LIN {X 0,Y 234.64,Z 487.256,A -85,B 0,C 180,E1 -19654.688,E2 -19654.688} C_VEL
LIN {X 0,Y 234.89,Z 487.224,A -85,B 0,C 180,E1 -19658.928,E2 -19658.928} C_VEL
LIN {X 0,Y 234.891,Z 487.223,A -85,B 0,C 180,E1 -19663.486,E2 -19663.486} C_VEL
LIN {X 0,Y 234.891,Z 487.226,A -85,B 0,C 180,E1 -19666.514,E2 -19666.514} C_VEL
LIN {X 0,Y 234.959,Z 487.213,A -85,B 0,C 180,E1 -19671.086,E2 -19671.086} C_VEL
LIN {X 0,Y 234.964,Z 487.215,A -85,B 0,C 180,E1 -19675.367,E2 -19675.367} C_VEL
LIN {X 0,Y 234.973,Z 487.214,A -85,B 0,C 180,E1 -19680.158,E2 -19680.158} C_VEL
LIN {X 0,Y 234.998,Z 487.212,A -85,B 0,C 180,E1 -19683.794,E2 -19683.794} C_VEL
LIN {X 0,Y 235.016,Z 487.206,A -85,B 0,C 180,E1 -19688.97,E2 -19688.97} C_VEL
LIN {X 0,Y 235.101,Z 487.198,A -85,B 0,C 180,E1 -19693.059,E2 -19693.059} C_VEL
LIN {X 0,Y 235.12,Z 487.195,A -85,B 0,C 180,E1 -19697.922,E2 -19697.922} C_VEL
LIN {X 0,Y 235.336,Z 487.169,A -85,B 0,C 180,E1 -19701.412,E2 -19701.412} C_VEL
LIN {X 0,Y 235.378,Z 487.163,A -85,B 0,C 180,E1 -19703.14,E2 -19703.14} C_VEL
LIN {X 0,Y 235.6,Z 487.138,A -85,B 0,C 180,E1 -19708.29,E2 -19708.29} C_VEL
LIN {X 0,Y 235.6,Z 487.138,A -85,B 0,C 180,E1 -19711.709,E2 -19711.709} C_VEL
LIN {X 0,Y 235.364,Z 487.164,A -85,B 0,C 180,E1 -19716.859,E2 -19716.859} C_VEL
LIN {X 0,Y 235.218,Z 487.184,A -85,B 0,C 180,E1 -19720.327,E2 -19720.327} C_VEL
LIN {X 0,Y 235.118,Z 487.196,A -85,B 0,C 180,E1 -19725.606,E2 -19725.606} C_VEL
LIN {X 0,Y 235.013,Z 487.209,A -85,B 0,C 180,E1 -19729.205,E2 -19729.205} C_VEL
LIN {X 0,Y 234.965,Z 487.212,A -85,B 0,C 180,E1 -19732.882,E2 -19732.882} C_VEL
LIN {X 0,Y 234.972,Z 487.214,A -85,B 0,C 180,E1 -19736.657,E2 -19736.657} C_VEL
LIN {X 0,Y 234.934,Z 487.215,A -85,B 0,C 180,E1 -19740.567,E2 -19740.567} C_VEL
LIN {X 0,Y 234.963,Z 487.215,A -85,B 0,C 180,E1 -19744.632,E2 -19744.632} C_VEL
LIN {X 0,Y 234.944,Z 487.215,A -85,B 0,C 180,E1 -19748.944,E2 -19748.944} C_VEL
LIN {X 0,Y 234.889,Z 487.226,A -85,B 0,C 180,E1 -19753.485,E2 -19753.485} C_VEL
LIN {X 0,Y 234.889,Z 487.223,A -85,B 0,C 180,E1 -19756.513,E2 -19756.513} C_VEL
LIN {X 0,Y 234.92,Z 487.22,A -85,B 0,C 180,E1 -19761.078,E2 -19761.078} C_VEL
LIN {X 0,Y 234.943,Z 487.219,A -85,B 0,C 180,E1 -19765.363,E2 -19765.363} C_VEL
LIN {X 0,Y 234.933,Z 487.22,A -85,B 0,C 180,E1 -19769.432,E2 -19769.432} C_VEL
LIN {X 0,Y 234.995,Z 487.212,A -85,B 0,C 180,E1 -19773.793,E2 -19773.793} C_VEL
LIN {X 0,Y 235.013,Z 487.209,A -85,B 0,C 180,E1 -19778.969,E2 -19778.969} C_VEL
LIN {X 0,Y 235.097,Z 487.198,A -85,B 0,C 180,E1 -19783.059,E2 -19783.059} C_VEL
LIN {X 0,Y 235.148,Z 487.194,A -85,B 0,C 180,E1 -19787.923,E2 -19787.923} C_VEL
LIN {X 0,Y 235.391,Z 487.164,A -85,B 0,C 180,E1 -19791.414,E2 -19791.414} C_VEL
LIN {X 0,Y 235.407,Z 487.159,A -85,B 0,C 180,E1 -19793.141,E2 -19793.141} C_VEL
LIN {X 0,Y 235.597,Z 487.136,A -85,B 0,C 180,E1 -19798.29,E2 -19798.29} C_VEL
LIN {X 0,Y 235.597,Z 487.136,A -85,B 0,C 180,E1 -19801.709,E2 -19801.709} C_VEL
LIN {X 0,Y 235.406,Z 487.16,A -85,B 0,C 180,E1 -19806.858,E2 -19806.858} C_VEL
LIN {X 0,Y 235.253,Z 487.176,A -85,B 0,C 180,E1 -19810.325,E2 -19810.325} C_VEL
LIN {X 0,Y 235.114,Z 487.199,A -85,B 0,C 180,E1 -19815.606,E2 -19815.606} C_VEL
LIN {X 0,Y 235.009,Z 487.21,A -85,B 0,C 180,E1 -19819.205,E2 -19819.205} C_VEL
LIN {X 0,Y 234.961,Z 487.216,A -85,B 0,C 180,E1 -19822.883,E2 -19822.883} C_VEL
LIN {X 0,Y 234.967,Z 487.214,A -85,B 0,C 180,E1 -19826.657,E2 -19826.657} C_VEL
LIN {X 0,Y 234.922,Z 487.219,A -85,B 0,C 180,E1 -19830.569,E2 -19830.569} C_VEL
LIN {X 0,Y 234.96,Z 487.215,A -85,B 0,C 180,E1 -19834.633,E2 -19834.633} C_VEL
LIN {X 0,Y 234.966,Z 487.214,A -85,B 0,C 180,E1 -19838.952,E2 -19838.952} C_VEL
LIN {X 0,Y 235.159,Z 487.364,A -85,B 0,C 180,E1 -19843.423,E2 -19843.423} C_VEL
LIN {X 0,Y 236.059,Z 492.395,A -85,B 0,C 180,E1 -19848.099,E2 -19848.099} C_VEL
LIN {X 0,Y 236.71,Z 496.121,A -85,B 0,C 180,E1 -19851.428,E2 -19851.428} C_VEL
LIN {X 0,Y 236.891,Z 498.627,A -85,B 0,C 180,E1 -19853.605,E2 -19853.605} C_VEL
LIN {X 0,Y 236.198,Z 501.988,A -85,B 0,C 180,E1 -19856.422,E2 -19856.422} C_VEL
LIN {X 0,Y 234.967,Z 507.976,A -85,B 0,C 180,E1 -19861.408,E2 -19861.408} C_VEL
LIN {X 0,Y 234.627,Z 509.787,A -85,B 0,C 180,E1 -19862.901,E2 -19862.901} C_VEL
LIN {X 0,Y 234.164,Z 511.237,A -85,B 0,C 180,E1 -19863.76,E2 -19863.76} C_VEL
LIN {X 0,Y 232.71,Z 514.431,A -85,B 0,C 180,E1 -19864.89,E2 -19864.89} C_VEL
LIN {X 0,Y 230.881,Z 518.451,A -85,B 0,C 180,E1 -19865.841,E2 -19865.841} C_VEL
LIN {X 0,Y 228.657,Z 524.846,A -85,B 0,C 180,E1 -19866.905,E2 -19866.905} C_VEL
LIN {X 0,Y 227.893,Z 530.135,A -85,B 0,C 180,E1 -19867.569,E2 -19867.569} C_VEL
LIN {X 0,Y 227.932,Z 531.961,A -85,B 0,C 180,E1 -19867.766,E2 -19867.766} C_VEL
LIN {X 0,Y 228.995,Z 545.084,A -85,B 0,C 180,E1 -19869.333,E2 -19869.333} C_VEL
LIN {X 0,Y 230.354,Z 558.222,A -85,B 0,C 180,E1 -19871.293,E2 -19871.293} C_VEL
LIN {X 0,Y 229.91,Z 564.614,A -85,B 0,C 180,E1 -19872.431,E2 -19872.431} C_VEL
LIN {X 0,Y 228.743,Z 574.152,A -85,B 0,C 180,E1 -19874.405,E2 -19874.405} C_VEL
LIN {X 0,Y 227.85,Z 583.066,A -85,B 0,C 180,E1 -19876.625,E2 -19876.625} C_VEL
LIN {X 0,Y 227.058,Z 591.816,A -85,B 0,C 180,E1 -19879.298,E2 -19879.298} C_VEL
LIN {X 0,Y 226.683,Z 598.895,A -85,B 0,C 180,E1 -19881.981,E2 -19881.981} C_VEL
LIN {X 0,Y 226.508,Z 604.521,A -85,B 0,C 180,E1 -19884.659,E2 -19884.659} C_VEL
LIN {X 0,Y 226.501,Z 608.915,A -85,B 0,C 180,E1 -19887.333,E2 -19887.333} C_VEL
LIN {X 0,Y 226.588,Z 612.194,A -85,B 0,C 180,E1 -19890,E2 -19890} C_VEL
LIN {X 0,Y 226.285,Z 613.769,A -85,B 0,C 180,E1 -19891.78,E2 -19891.78} C_VEL
LIN {X 0,Y 225.922,Z 615.651,A -85,B 0,C 180,E1 -19895.355,E2 -19895.355} C_VEL
LIN {X 0,Y 226.153,Z 616.056,A -85,B 0,C 180,E1 -19898.939,E2 -19898.939} C_VEL
LIN {X 0,Y 227.195,Z 615.063,A -85,B 0,C 180,E1 -19902.506,E2 -19902.506} C_VEL
LIN {X 0,Y 229.251,Z 612.694,A -85,B 0,C 180,E1 -19906.017,E2 -19906.017} C_VEL
LIN {X 0,Y 232.384,Z 608.934,A -85,B 0,C 180,E1 -19909.432,E2 -19909.432} C_VEL
LIN {X 0,Y 236.369,Z 603.761,A -85,B 0,C 180,E1 -19912.739,E2 -19912.739} C_VEL
LIN {X 0,Y 240.175,Z 598.876,A -85,B 0,C 180,E1 -19915.107,E2 -19915.107} C_VEL
LIN {X 0,Y 246.115,Z 590.937,A -85,B 0,C 180,E1 -19918.111,E2 -19918.111} C_VEL
LIN {X 0,Y 251.032,Z 583.774,A -85,B 0,C 180,E1 -19920.261,E2 -19920.261} C_VEL
LIN {X 0,Y 253.685,Z 578.77,A -85,B 0,C 180,E1 -19921.761,E2 -19921.761} C_VEL
LIN {X 0,Y 256.161,Z 572.028,A -85,B 0,C 180,E1 -19923.971,E2 -19923.971} C_VEL
LIN {X 0,Y 258.198,Z 564.336,A -85,B 0,C 180,E1 -19926.786,E2 -19926.786} C_VEL
LIN {X 0,Y 259.165,Z 560.003,A -85,B 0,C 180,E1 -19928.588,E2 -19928.588} C_VEL
LIN {X 0,Y 259.899,Z 556.273,A -85,B 0,C 180,E1 -19930.466,E2 -19930.466} C_VEL
LIN {X 0,Y 260.12,Z 553.505,A -85,B 0,C 180,E1 -19932.49,E2 -19932.49} C_VEL
LIN {X 0,Y 260.395,Z 551.497,A -85,B 0,C 180,E1 -19934.567,E2 -19934.567} C_VEL
LIN {X 0,Y 260.509,Z 550.609,A -85,B 0,C 180,E1 -19936.754,E2 -19936.754} C_VEL
LIN {X 0,Y 260.631,Z 551.068,A -85,B 0,C 180,E1 -19939.672,E2 -19939.672} C_VEL
LIN {X 0,Y 260.998,Z 552.105,A -85,B 0,C 180,E1 -19941.733,E2 -19941.733} C_VEL
LIN {X 0,Y 261.38,Z 553.873,A -85,B 0,C 180,E1 -19943.77,E2 -19943.77} C_VEL
LIN {X 0,Y 261.44,Z 557.559,A -85,B 0,C 180,E1 -19946.444,E2 -19946.444} C_VEL
LIN {X 0,Y 260.967,Z 561.356,A -85,B 0,C 180,E1 -19948.526,E2 -19948.526} C_VEL
LIN {X 0,Y 260.113,Z 563.075,A -85,B 0,C 180,E1 -19949.112,E2 -19949.112} C_VEL
LIN {X 0,Y 253.924,Z 571.515,A -85,B 0,C 180,E1 -19951.482,E2 -19951.482} C_VEL
LIN {X 0,Y 248.247,Z 578.439,A -85,B 0,C 180,E1 -19953.972,E2 -19953.972} C_VEL
LIN {X 0,Y 243.868,Z 583.268,A -85,B 0,C 180,E1 -19956.205,E2 -19956.205} C_VEL
LIN {X 0,Y 238.859,Z 588.281,A -85,B 0,C 180,E1 -19959.325,E2 -19959.325} C_VEL
LIN {X 0,Y 234.733,Z 591.746,A -85,B 0,C 180,E1 -19962.579,E2 -19962.579} C_VEL
LIN {X 0,Y 232.898,Z 592.963,A -85,B 0,C 180,E1 -19964.242,E2 -19964.242} C_VEL
LIN {X 0,Y 230.124,Z 594.323,A -85,B 0,C 180,E1 -19967.656,E2 -19967.656} C_VEL
LIN {X 0,Y 227.906,Z 594.264,A -85,B 0,C 180,E1 -19971.131,E2 -19971.131} C_VEL
LIN {X 0,Y 226.816,Z 592.766,A -85,B 0,C 180,E1 -19974.667,E2 -19974.667} C_VEL
LIN {X 0,Y 226.416,Z 591.482,A -85,B 0,C 180,E1 -19976.441,E2 -19976.441} C_VEL
LIN {X 0,Y 225.976,Z 587.71,A -85,B 0,C 180,E1 -19980,E2 -19980} C_VEL
LIN {X 0,Y 225.999,Z 583.818,A -85,B 0,C 180,E1 -19982.674,E2 -19982.674} C_VEL
LIN {X 0,Y 226.077,Z 578.823,A -85,B 0,C 180,E1 -19985.352,E2 -19985.352} C_VEL
LIN {X 0,Y 226.624,Z 571.523,A -85,B 0,C 180,E1 -19988.471,E2 -19988.471} C_VEL
LIN {X 0,Y 227.301,Z 563.747,A -85,B 0,C 180,E1 -19991.143,E2 -19991.143} C_VEL
LIN {X 0,Y 228.272,Z 554.253,A -85,B 0,C 180,E1 -19993.805,E2 -19993.805} C_VEL
LIN {X 0,Y 229.552,Z 543.626,A -85,B 0,C 180,E1 -19996.223,E2 -19996.223} C_VEL
LIN {X 0,Y 230.933,Z 531.732,A -85,B 0,C 180,E1 -19998.406,E2 -19998.406} C_VEL
LIN {X 0,Y 232.048,Z 520.174,A -85,B 0,C 180,E1 -20000.133,E2 -20000.133} C_VEL
LIN {X 0,Y 229.504,Z 506.121,A -85,B 0,C 180,E1 -20001.896,E2 -20001.896} C_VEL
LIN {X 0,Y 227.192,Z 492.743,A -85,B 0,C 180,E1 -20003.213,E2 -20003.213} C_VEL
LIN {X 0,Y 226.512,Z 488.273,A -85,B 0,C 180,E1 -20003.585,E2 -20003.585} C_VEL
LIN {X 0,Y 226.902,Z 488.224,A -85,B 0,C 180,E1 -20007.685,E2 -20007.685} C_VEL
LIN {X 0,Y 227.31,Z 488.167,A -85,B 0,C 180,E1 -20011.71,E2 -20011.71} C_VEL
LIN {X 0,Y 227.698,Z 488.121,A -85,B 0,C 180,E1 -20015.906,E2 -20015.906} C_VEL
LIN {X 0,Y 227.817,Z 488.105,A -85,B 0,C 180,E1 -20019.535,E2 -20019.535} C_VEL
LIN {X 0,Y 227.812,Z 488.105,A -85,B 0,C 180,E1 -20022.743,E2 -20022.743} C_VEL
LIN {X 0,Y 227.818,Z 488.105,A -85,B 0,C 180,E1 -20027.259,E2 -20027.259} C_VEL
LIN {X 0,Y 227.873,Z 488.098,A -85,B 0,C 180,E1 -20031.914,E2 -20031.914} C_VEL
LIN {X 0,Y 227.893,Z 488.097,A -85,B 0,C 180,E1 -20036.373,E2 -20036.373} C_VEL
LIN {X 0,Y 227.923,Z 488.093,A -85,B 0,C 180,E1 -20040.438,E2 -20040.438} C_VEL
LIN {X 0,Y 227.933,Z 488.092,A -85,B 0,C 180,E1 -20044.426,E2 -20044.426} C_VEL
LIN {X 0,Y 227.967,Z 488.087,A -85,B 0,C 180,E1 -20048.287,E2 -20048.287} C_VEL
LIN {X 0,Y 228.04,Z 488.078,A -85,B 0,C 180,E1 -20052.825,E2 -20052.825} C_VEL
LIN {X 0,Y 228.078,Z 488.07,A -85,B 0,C 180,E1 -20057.543,E2 -20057.543} C_VEL
LIN {X 0,Y 228.272,Z 488.048,A -85,B 0,C 180,E1 -20061.144,E2 -20061.144} C_VEL
LIN {X 0,Y 228.329,Z 488.041,A -85,B 0,C 180,E1 -20062.927,E2 -20062.927} C_VEL
LIN {X 0,Y 228.559,Z 488.015,A -85,B 0,C 180,E1 -20068.238,E2 -20068.238} C_VEL
LIN {X 0,Y 228.558,Z 488.015,A -85,B 0,C 180,E1 -20071.762,E2 -20071.762} C_VEL
LIN {X 0,Y 228.316,Z 488.042,A -85,B 0,C 180,E1 -20077.072,E2 -20077.072} C_VEL
LIN {X 0,Y 228.15,Z 488.063,A -85,B 0,C 180,E1 -20080.651,E2 -20080.651} C_VEL
LIN {X 0,Y 228.069,Z 488.074,A -85,B 0,C 180,E1 -20084.271,E2 -20084.271} C_VEL
LIN {X 0,Y 228.007,Z 488.085,A -85,B 0,C 180,E1 -20087.953,E2 -20087.953} C_VEL
LIN {X 0,Y 227.934,Z 488.089,A -85,B 0,C 180,E1 -20092.329,E2 -20092.329} C_VEL
LIN {X 0,Y 227.946,Z 488.089,A -85,B 0,C 180,E1 -20096.602,E2 -20096.602} C_VEL
LIN {X 0,Y 227.911,Z 488.091,A -85,B 0,C 180,E1 -20100.295,E2 -20100.295} C_VEL
LIN {X 0,Y 227.893,Z 488.098,A -85,B 0,C 180,E1 -20103.717,E2 -20103.717} C_VEL
LIN {X 0,Y 227.872,Z 488.098,A -85,B 0,C 180,E1 -20108.085,E2 -20108.085} C_VEL
LIN {X 0,Y 227.816,Z 488.105,A -85,B 0,C 180,E1 -20112.741,E2 -20112.741} C_VEL
LIN {X 0,Y 227.812,Z 488.105,A -85,B 0,C 180,E1 -20117.257,E2 -20117.257} C_VEL
LIN {X 0,Y 227.846,Z 488.104,A -85,B 0,C 180,E1 -20121.908,E2 -20121.908} C_VEL
LIN {X 0,Y 227.884,Z 488.094,A -85,B 0,C 180,E1 -20126.375,E2 -20126.375} C_VEL
LIN {X 0,Y 227.921,Z 488.092,A -85,B 0,C 180,E1 -20130.437,E2 -20130.437} C_VEL
LIN {X 0,Y 227.93,Z 488.089,A -85,B 0,C 180,E1 -20134.425,E2 -20134.425} C_VEL
LIN {X 0,Y 227.963,Z 488.087,A -85,B 0,C 180,E1 -20138.287,E2 -20138.287} C_VEL
LIN {X 0,Y 228.036,Z 488.077,A -85,B 0,C 180,E1 -20142.825,E2 -20142.825} C_VEL
LIN {X 0,Y 228.095,Z 488.073,A -85,B 0,C 180,E1 -20147.544,E2 -20147.544} C_VEL
LIN {X 0,Y 228.326,Z 488.043,A -85,B 0,C 180,E1 -20151.146,E2 -20151.146} C_VEL
LIN {X 0,Y 228.359,Z 488.036,A -85,B 0,C 180,E1 -20152.928,E2 -20152.928} C_VEL
LIN {X 0,Y 228.556,Z 488.013,A -85,B 0,C 180,E1 -20158.237,E2 -20158.237} C_VEL
LIN {X 0,Y 228.555,Z 488.012,A -85,B 0,C 180,E1 -20161.762,E2 -20161.762} C_VEL
LIN {X 0,Y 228.359,Z 488.039,A -85,B 0,C 180,E1 -20167.071,E2 -20167.071} C_VEL
LIN {X 0,Y 228.172,Z 488.058,A -85,B 0,C 180,E1 -20170.65,E2 -20170.65} C_VEL
LIN {X 0,Y 228.058,Z 488.075,A -85,B 0,C 180,E1 -20176.102,E2 -20176.102} C_VEL
LIN {X 0,Y 227.943,Z 488.088,A -85,B 0,C 180,E1 -20179.825,E2 -20179.825} C_VEL
LIN {X 0,Y 227.914,Z 488.095,A -85,B 0,C 180,E1 -20183.632,E2 -20183.632} C_VEL
LIN {X 0,Y 227.879,Z 488.097,A -85,B 0,C 180,E1 -20187.556,E2 -20187.556} C_VEL
LIN {X 0,Y 227.869,Z 488.101,A -85,B 0,C 180,E1 -20191.622,E2 -20191.622} C_VEL
LIN {X 0,Y 227.901,Z 488.093,A -85,B 0,C 180,E1 -20195.868,E2 -20195.868} C_VEL
LIN {X 0,Y 227.916,Z 488.092,A -85,B 0,C 180,E1 -20200.357,E2 -20200.357} C_VEL
LIN {X 0,Y 228.11,Z 488.177,A -85,B 0,C 180,E1 -20203.428,E2 -20203.428} C_VEL
LIN {X 0,Y 229.108,Z 493.726,A -85,B 0,C 180,E1 -20208.737,E2 -20208.737} C_VEL
LIN {X 0,Y 229.739,Z 497.598,A -85,B 0,C 180,E1 -20212.279,E2 -20212.279} C_VEL
LIN {X 0,Y 229.664,Z 500.056,A -85,B 0,C 180,E1 -20214.45,E2 -20214.45} C_VEL
LIN {X 0,Y 228.276,Z 505.955,A -85,B 0,C 180,E1 -20219.546,E2 -20219.546} C_VEL
LIN {X 0,Y 227.217,Z 511.521,A -85,B 0,C 180,E1 -20224.34,E2 -20224.34} C_VEL
LIN {X 0,Y 226.937,Z 513.601,A -85,B 0,C 180,E1 -20226.139,E2 -20226.139} C_VEL
LIN {X 0,Y 227.507,Z 526.824,A -85,B 0,C 180,E1 -20227.248,E2 -20227.248} C_VEL
LIN {X 0,Y 227.932,Z 531.961,A -85,B 0,C 180,E1 -20227.766,E2 -20227.766} C_VEL
LIN {X 0,Y 227.751,Z 537.377,A -85,B 0,C 180,E1 -20228.353,E2 -20228.353} C_VEL
LIN {X 0,Y 225.867,Z 546.084,A -85,B 0,C 180,E1 -20229.434,E2 -20229.434} C_VEL
LIN {X 0,Y 224.113,Z 552.813,A -85,B 0,C 180,E1 -20230.42,E2 -20230.42} C_VEL
LIN {X 0,Y 223.29,Z 559.395,A -85,B 0,C 180,E1 -20231.529,E2 -20231.529} C_VEL
LIN {X 0,Y 222.075,Z 570.338,A -85,B 0,C 180,E1 -20233.688,E2 -20233.688} C_VEL
LIN {X 0,Y 221.162,Z 578.904,A -85,B 0,C 180,E1 -20235.743,E2 -20235.743} C_VEL
LIN {X 0,Y 220.241,Z 588.254,A -85,B 0,C 180,E1 -20238.496,E2 -20238.496} C_VEL
LIN {X 0,Y 219.779,Z 595.885,A -85,B 0,C 180,E1 -20241.264,E2 -20241.264} C_VEL
LIN {X 0,Y 219.564,Z 601.199,A -85,B 0,C 180,E1 -20243.626,E2 -20243.626} C_VEL
LIN {X 0,Y 219.505,Z 606.125,A -85,B 0,C 180,E1 -20246.329,E2 -20246.329} C_VEL
LIN {X 0,Y 219.528,Z 609.978,A -85,B 0,C 180,E1 -20249.083,E2 -20249.083} C_VEL
LIN {X 0,Y 219.571,Z 611.024,A -85,B 0,C 180,E1 -20250,E2 -20250} C_VEL
LIN {X 0,Y 219.273,Z 612.679,A -85,B 0,C 180,E1 -20251.837,E2 -20251.837} C_VEL
LIN {X 0,Y 218.886,Z 614.828,A -85,B 0,C 180,E1 -20255.528,E2 -20255.528} C_VEL
LIN {X 0,Y 219.122,Z 615.516,A -85,B 0,C 180,E1 -20259.229,E2 -20259.229} C_VEL
LIN {X 0,Y 220.227,Z 614.78,A -85,B 0,C 180,E1 -20262.909,E2 -20262.909} C_VEL
LIN {X 0,Y 222.43,Z 612.714,A -85,B 0,C 180,E1 -20266.522,E2 -20266.522} C_VEL
LIN {X 0,Y 225.697,Z 609.304,A -85,B 0,C 180,E1 -20270.032,E2 -20270.032} C_VEL
LIN {X 0,Y 228.769,Z 605.774,A -85,B 0,C 180,E1 -20272.65,E2 -20272.65} C_VEL
LIN {X 0,Y 233.847,Z 599.995,A -85,B 0,C 180,E1 -20275.835,E2 -20275.835} C_VEL
LIN {X 0,Y 240.003,Z 592.536,A -85,B 0,C 180,E1 -20278.893,E2 -20278.893} C_VEL
LIN {X 0,Y 245.955,Z 584.69,A -85,B 0,C 180,E1 -20281.432,E2 -20281.432} C_VEL
LIN {X 0,Y 248.034,Z 581.14,A -85,B 0,C 180,E1 -20282.573,E2 -20282.573} C_VEL
LIN {X 0,Y 251.092,Z 574.057,A -85,B 0,C 180,E1 -20285.116,E2 -20285.116} C_VEL
LIN {X 0,Y 253.186,Z 567.758,A -85,B 0,C 180,E1 -20287.639,E2 -20287.639} C_VEL
LIN {X 0,Y 254.692,Z 562.719,A -85,B 0,C 180,E1 -20289.973,E2 -20289.973} C_VEL
LIN {X 0,Y 255.329,Z 559.621,A -85,B 0,C 180,E1 -20291.997,E2 -20291.997} C_VEL
LIN {X 0,Y 255.734,Z 557.187,A -85,B 0,C 180,E1 -20294.396,E2 -20294.396} C_VEL
LIN {X 0,Y 255.891,Z 556.401,A -85,B 0,C 180,E1 -20295.569,E2 -20295.569} C_VEL
LIN {X 0,Y 255.916,Z 556.066,A -85,B 0,C 180,E1 -20297.858,E2 -20297.858} C_VEL
LIN {X 0,Y 256.097,Z 556.948,A -85,B 0,C 180,E1 -20300.863,E2 -20300.863} C_VEL
LIN {X 0,Y 256.424,Z 559.105,A -85,B 0,C 180,E1 -20303.786,E2 -20303.786} C_VEL
LIN {X 0,Y 256.22,Z 561.053,A -85,B 0,C 180,E1 -20305.376,E2 -20305.376} C_VEL
LIN {X 0,Y 255.688,Z 564.505,A -85,B 0,C 180,E1 -20307.604,E2 -20307.604} C_VEL
LIN {X 0,Y 254.553,Z 566.48,A -85,B 0,C 180,E1 -20308.361,E2 -20308.361} C_VEL
LIN {X 0,Y 248.104,Z 574.414,A -85,B 0,C 180,E1 -20310.749,E2 -20310.749} C_VEL
LIN {X 0,Y 242.187,Z 580.835,A -85,B 0,C 180,E1 -20313.27,E2 -20313.27} C_VEL
LIN {X 0,Y 237.65,Z 585.299,A -85,B 0,C 180,E1 -20315.543,E2 -20315.543} C_VEL
LIN {X 0,Y 232.418,Z 589.853,A -85,B 0,C 180,E1 -20318.724,E2 -20318.724} C_VEL
LIN {X 0,Y 228.076,Z 592.969,A -85,B 0,C 180,E1 -20322.053,E2 -20322.053} C_VEL
LIN {X 0,Y 226.164,Z 594.008,A -85,B 0,C 180,E1 -20323.76,E2 -20323.76} C_VEL
LIN {X 0,Y 223.231,Z 595.007,A -85,B 0,C 180,E1 -20327.269,E2 -20327.269} C_VEL
LIN {X 0,Y 220.919,Z 594.665,A -85,B 0,C 180,E1 -20330.848,E2 -20330.848} C_VEL
LIN {X 0,Y 219.754,Z 592.868,A -85,B 0,C 180,E1 -20334.495,E2 -20334.495} C_VEL
LIN {X 0,Y 219.052,Z 589.599,A -85,B 0,C 180,E1 -20338.162,E2 -20338.162} C_VEL
LIN {X 0,Y 218.882,Z 586.103,A -85,B 0,C 180,E1 -20340.92,E2 -20340.92} C_VEL
LIN {X 0,Y 218.927,Z 581.625,A -85,B 0,C 180,E1 -20343.682,E2 -20343.682} C_VEL
LIN {X 0,Y 219.256,Z 575.022,A -85,B 0,C 180,E1 -20346.904,E2 -20346.904} C_VEL
LIN {X 0,Y 219.771,Z 567.895,A -85,B 0,C 180,E1 -20349.666,E2 -20349.666} C_VEL
LIN {X 0,Y 220.639,Z 559.205,A -85,B 0,C 180,E1 -20352.416,E2 -20352.416} C_VEL
LIN {X 0,Y 221.802,Z 548.64,A -85,B 0,C 180,E1 -20355.154,E2 -20355.154} C_VEL
LIN {X 0,Y 223.056,Z 537.863,A -85,B 0,C 180,E1 -20357.418,E2 -20357.418} C_VEL
LIN {X 0,Y 224.215,Z 527.534,A -85,B 0,C 180,E1 -20359.216,E2 -20359.216} C_VEL
LIN {X 0,Y 224.842,Z 520.022,A -85,B 0,C 180,E1 -20360.325,E2 -20360.325} C_VEL
LIN {X 0,Y 222.45,Z 506.821,A -85,B 0,C 180,E1 -20362.035,E2 -20362.035} C_VEL
LIN {X 0,Y 220.202,Z 493.731,A -85,B 0,C 180,E1 -20363.374,E2 -20363.374} C_VEL
LIN {X 0,Y 219.505,Z 489.147,A -85,B 0,C 180,E1 -20363.777,E2 -20363.777} C_VEL
LIN {X 0,Y 219.951,Z 489.087,A -85,B 0,C 180,E1 -20368.64,E2 -20368.64} C_VEL
LIN {X 0,Y 220.361,Z 489.031,A -85,B 0,C 180,E1 -20372.833,E2 -20372.833} C_VEL
LIN {X 0,Y 220.711,Z 488.99,A -85,B 0,C 180,E1 -20377.243,E2 -20377.243} C_VEL
LIN {X 0,Y 220.776,Z 488.984,A -85,B 0,C 180,E1 -20380.182,E2 -20380.182} C_VEL
LIN {X 0,Y 220.777,Z 488.985,A -85,B 0,C 180,E1 -20384.454,E2 -20384.454} C_VEL
LIN {X 0,Y 220.779,Z 488.984,A -85,B 0,C 180,E1 -20388.049,E2 -20388.049} C_VEL
LIN {X 0,Y 220.835,Z 488.975,A -85,B 0,C 180,E1 -20392.794,E2 -20392.794} C_VEL
LIN {X 0,Y 220.828,Z 488.975,A -85,B 0,C 180,E1 -20397.245,E2 -20397.245} C_VEL
LIN {X 0,Y 220.84,Z 488.973,A -85,B 0,C 180,E1 -20401.486,E2 -20401.486} C_VEL
LIN {X 0,Y 220.872,Z 488.971,A -85,B 0,C 180,E1 -20405.565,E2 -20405.565} C_VEL
LIN {X 0,Y 220.898,Z 488.965,A -85,B 0,C 180,E1 -20409.514,E2 -20409.514} C_VEL
LIN {X 0,Y 221.021,Z 488.952,A -85,B 0,C 180,E1 -20413.37,E2 -20413.37} C_VEL
LIN {X 0,Y 221.086,Z 488.943,A -85,B 0,C 180,E1 -20419.004,E2 -20419.004} C_VEL
LIN {X 0,Y 221.264,Z 488.921,A -85,B 0,C 180,E1 -20422.7,E2 -20422.7} C_VEL
LIN {X 0,Y 221.517,Z 488.893,A -85,B 0,C 180,E1 -20428.181,E2 -20428.181} C_VEL
LIN {X 0,Y 221.516,Z 488.893,A -85,B 0,C 180,E1 -20431.818,E2 -20431.818} C_VEL
LIN {X 0,Y 221.253,Z 488.923,A -85,B 0,C 180,E1 -20437.299,E2 -20437.299} C_VEL
LIN {X 0,Y 221.086,Z 488.943,A -85,B 0,C 180,E1 -20440.995,E2 -20440.995} C_VEL
LIN {X 0,Y 221.021,Z 488.952,A -85,B 0,C 180,E1 -20446.629,E2 -20446.629} C_VEL
LIN {X 0,Y 220.897,Z 488.966,A -85,B 0,C 180,E1 -20450.485,E2 -20450.485} C_VEL
LIN {X 0,Y 220.871,Z 488.971,A -85,B 0,C 180,E1 -20454.434,E2 -20454.434} C_VEL
LIN {X 0,Y 220.839,Z 488.974,A -85,B 0,C 180,E1 -20458.513,E2 -20458.513} C_VEL
LIN {X 0,Y 220.827,Z 488.975,A -85,B 0,C 180,E1 -20462.754,E2 -20462.754} C_VEL
LIN {X 0,Y 220.84,Z 488.975,A -85,B 0,C 180,E1 -20467.287,E2 -20467.287} C_VEL
LIN {X 0,Y 220.777,Z 488.985,A -85,B 0,C 180,E1 -20471.951,E2 -20471.951} C_VEL
LIN {X 0,Y 220.775,Z 488.985,A -85,B 0,C 180,E1 -20475.545,E2 -20475.545} C_VEL
LIN {X 0,Y 220.808,Z 488.978,A -85,B 0,C 180,E1 -20480.462,E2 -20480.462} C_VEL
LIN {X 0,Y 220.805,Z 488.978,A -85,B 0,C 180,E1 -20485.045,E2 -20485.045} C_VEL
LIN {X 0,Y 220.869,Z 488.971,A -85,B 0,C 180,E1 -20489.394,E2 -20489.394} C_VEL
LIN {X 0,Y 220.897,Z 488.97,A -85,B 0,C 180,E1 -20493.549,E2 -20493.549} C_VEL
LIN {X 0,Y 220.879,Z 488.97,A -85,B 0,C 180,E1 -20497.553,E2 -20497.553} C_VEL
LIN {X 0,Y 220.985,Z 488.955,A -85,B 0,C 180,E1 -20502.57,E2 -20502.57} C_VEL
LIN {X 0,Y 221.027,Z 488.951,A -85,B 0,C 180,E1 -20507.139,E2 -20507.139} C_VEL
LIN {X 0,Y 221.259,Z 488.922,A -85,B 0,C 180,E1 -20510.861,E2 -20510.861} C_VEL
LIN {X 0,Y 221.312,Z 488.913,A -85,B 0,C 180,E1 -20512.702,E2 -20512.702} C_VEL
LIN {X 0,Y 221.514,Z 488.891,A -85,B 0,C 180,E1 -20518.181,E2 -20518.181} C_VEL
LIN {X 0,Y 221.513,Z 488.889,A -85,B 0,C 180,E1 -20521.818,E2 -20521.818} C_VEL
LIN {X 0,Y 221.312,Z 488.918,A -85,B 0,C 180,E1 -20527.297,E2 -20527.297} C_VEL
LIN {X 0,Y 221.117,Z 488.938,A -85,B 0,C 180,E1 -20530.994,E2 -20530.994} C_VEL
LIN {X 0,Y 221.016,Z 488.952,A -85,B 0,C 180,E1 -20536.629,E2 -20536.629} C_VEL
LIN {X 0,Y 220.893,Z 488.965,A -85,B 0,C 180,E1 -20540.486,E2 -20540.486} C_VEL
LIN {X 0,Y 220.867,Z 488.971,A -85,B 0,C 180,E1 -20544.435,E2 -20544.435} C_VEL
LIN {X 0,Y 220.826,Z 488.972,A -85,B 0,C 180,E1 -20548.515,E2 -20548.515} C_VEL
LIN {X 0,Y 220.823,Z 488.977,A -85,B 0,C 180,E1 -20552.755,E2 -20552.755} C_VEL
LIN {X 0,Y 220.838,Z 488.974,A -85,B 0,C 180,E1 -20557.288,E2 -20557.288} C_VEL
LIN {X 0,Y 220.947,Z 488.961,A -85,B 0,C 180,E1 -20561.911,E2 -20561.911} C_VEL
LIN {X 0,Y 221.085,Z 489.124,A -85,B 0,C 180,E1 -20563.599,E2 -20563.599} C_VEL
LIN {X 0,Y 221.932,Z 493.899,A -85,B 0,C 180,E1 -20568.317,E2 -20568.317} C_VEL
LIN {X 0,Y 222.644,Z 497.881,A -85,B 0,C 180,E1 -20572.106,E2 -20572.106} C_VEL
LIN {X 0,Y 222.604,Z 500.243,A -85,B 0,C 180,E1 -20574.264,E2 -20574.264} C_VEL
LIN {X 0,Y 221.199,Z 506.017,A -85,B 0,C 180,E1 -20579.446,E2 -20579.446} C_VEL
LIN {X 0,Y 220.099,Z 511.617,A -85,B 0,C 180,E1 -20584.465,E2 -20584.465} C_VEL
LIN {X 0,Y 219.849,Z 513.48,A -85,B 0,C 180,E1 -20585.948,E2 -20585.948} C_VEL
LIN {X 0,Y 220.442,Z 527.242,A -85,B 0,C 180,E1 -20587.137,E2 -20587.137} C_VEL
LIN {X 0,Y 221.545,Z 541.001,A -85,B 0,C 180,E1 -20588.726,E2 -20588.726} C_VEL
LIN {X 0,Y 222.691,Z 553.141,A -85,B 0,C 180,E1 -20590.473,E2 -20590.473} C_VEL
LIN {X 0,Y 223.29,Z 559.395,A -85,B 0,C 180,E1 -20591.529,E2 -20591.529} C_VEL
LIN {X 0,Y 222.89,Z 562.631,A -85,B 0,C 180,E1 -20592.117,E2 -20592.117} C_VEL
LIN {X 0,Y 221.851,Z 565.638,A -85,B 0,C 180,E1 -20592.714,E2 -20592.714} C_VEL
LIN {X 0,Y 218.723,Z 571.21,A -85,B 0,C 180,E1 -20593.956,E2 -20593.956} C_VEL
LIN {X 0,Y 214.845,Z 577.728,A -85,B 0,C 180,E1 -20595.68,E2 -20595.68} C_VEL
LIN {X 0,Y 213.753,Z 581.686,A -85,B 0,C 180,E1 -20596.824,E2 -20596.824} C_VEL
LIN {X 0,Y 213.012,Z 590.102,A -85,B 0,C 180,E1 -20599.545,E2 -20599.545} C_VEL
LIN {X 0,Y 212.645,Z 597.527,A -85,B 0,C 180,E1 -20602.528,E2 -20602.528} C_VEL
LIN {X 0,Y 212.526,Z 602.962,A -85,B 0,C 180,E1 -20605.258,E2 -20605.258} C_VEL
LIN {X 0,Y 212.537,Z 607.396,A -85,B 0,C 180,E1 -20608.105,E2 -20608.105} C_VEL
LIN {X 0,Y 212.572,Z 609.731,A -85,B 0,C 180,E1 -20610,E2 -20610} C_VEL
LIN {X 0,Y 212.258,Z 611.558,A -85,B 0,C 180,E1 -20611.898,E2 -20611.898} C_VEL
LIN {X 0,Y 211.849,Z 613.936,A -85,B 0,C 180,E1 -20615.712,E2 -20615.712} C_VEL
LIN {X 0,Y 212.111,Z 614.863,A -85,B 0,C 180,E1 -20619.537,E2 -20619.537} C_VEL
LIN {X 0,Y 213.274,Z 614.441,A -85,B 0,C 180,E1 -20623.337,E2 -20623.337} C_VEL
LIN {X 0,Y 215.631,Z 612.708,A -85,B 0,C 180,E1 -20627.058,E2 -20627.058} C_VEL
LIN {X 0,Y 219.038,Z 609.647,A -85,B 0,C 180,E1 -20630.668,E2 -20630.668} C_VEL
LIN {X 0,Y 223.434,Z 605.246,A -85,B 0,C 180,E1 -20634.137,E2 -20634.137} C_VEL
LIN {X 0,Y 229.087,Z 599.459,A -85,B 0,C 180,E1 -20637.399,E2 -20637.399} C_VEL
LIN {X 0,Y 235.727,Z 592.146,A -85,B 0,C 180,E1 -20640.454,E2 -20640.454} C_VEL
LIN {X 0,Y 240.966,Z 585.652,A -85,B 0,C 180,E1 -20642.655,E2 -20642.655} C_VEL
LIN {X 0,Y 243.013,Z 582.425,A -85,B 0,C 180,E1 -20643.83,E2 -20643.83} C_VEL
LIN {X 0,Y 245.962,Z 576.319,A -85,B 0,C 180,E1 -20646.228,E2 -20646.228} C_VEL
LIN {X 0,Y 248.574,Z 569.996,A -85,B 0,C 180,E1 -20649.034,E2 -20649.034} C_VEL
LIN {X 0,Y 249.904,Z 566.189,A -85,B 0,C 180,E1 -20651.084,E2 -20651.084} C_VEL
LIN {X 0,Y 250.579,Z 563.606,A -85,B 0,C 180,E1 -20653.179,E2 -20653.179} C_VEL
LIN {X 0,Y 251.108,Z 561.681,A -85,B 0,C 180,E1 -20655.597,E2 -20655.597} C_VEL
LIN {X 0,Y 251.149,Z 561.304,A -85,B 0,C 180,E1 -20657.809,E2 -20657.809} C_VEL
LIN {X 0,Y 251.112,Z 561.753,A -85,B 0,C 180,E1 -20659.931,E2 -20659.931} C_VEL
LIN {X 0,Y 251.189,Z 562.768,A -85,B 0,C 180,E1 -20662.009,E2 -20662.009} C_VEL
LIN {X 0,Y 251.115,Z 564.632,A -85,B 0,C 180,E1 -20664.256,E2 -20664.256} C_VEL
LIN {X 0,Y 250.325,Z 567.978,A -85,B 0,C 180,E1 -20666.806,E2 -20666.806} C_VEL
LIN {X 0,Y 249.007,Z 569.901,A -85,B 0,C 180,E1 -20667.571,E2 -20667.571} C_VEL
LIN {X 0,Y 241.396,Z 578.168,A -85,B 0,C 180,E1 -20670.335,E2 -20670.335} C_VEL
LIN {X 0,Y 236.16,Z 583.177,A -85,B 0,C 180,E1 -20672.531,E2 -20672.531} C_VEL
LIN {X 0,Y 230.029,Z 588.425,A -85,B 0,C 180,E1 -20675.641,E2 -20675.641} C_VEL
LIN {X 0,Y 225.975,Z 591.397,A -85,B 0,C 180,E1 -20678.087,E2 -20678.087} C_VEL
LIN {X 0,Y 221.43,Z 594.12,A -85,B 0,C 180,E1 -20681.495,E2 -20681.495} C_VEL
LIN {X 0,Y 217.798,Z 595.488,A -85,B 0,C 180,E1 -20685.04,E2 -20685.04} C_VEL
LIN {X 0,Y 214.981,Z 595.507,A -85,B 0,C 180,E1 -20688.689,E2 -20688.689} C_VEL
LIN {X 0,Y 213.193,Z 594.104,A -85,B 0,C 180,E1 -20692.423,E2 -20692.423} C_VEL
LIN {X 0,Y 212.301,Z 591.302,A -85,B 0,C 180,E1 -20696.204,E2 -20696.204} C_VEL
LIN {X 0,Y 211.879,Z 588.198,A -85,B 0,C 180,E1 -20699.05,E2 -20699.05} C_VEL
LIN {X 0,Y 211.85,Z 584.159,A -85,B 0,C 180,E1 -20701.902,E2 -20701.902} C_VEL
LIN {X 0,Y 211.919,Z 578.532,A -85,B 0,C 180,E1 -20705.023,E2 -20705.023} C_VEL
LIN {X 0,Y 212.394,Z 571.648,A -85,B 0,C 180,E1 -20708.085,E2 -20708.085} C_VEL
LIN {X 0,Y 213.193,Z 562.296,A -85,B 0,C 180,E1 -20711.408,E2 -20711.408} C_VEL
LIN {X 0,Y 214.048,Z 554.113,A -85,B 0,C 180,E1 -20713.772,E2 -20713.772} C_VEL
LIN {X 0,Y 215.37,Z 543.318,A -85,B 0,C 180,E1 -20716.347,E2 -20716.347} C_VEL
LIN {X 0,Y 216.798,Z 531.37,A -85,B 0,C 180,E1 -20718.671,E2 -20718.671} C_VEL
LIN {X 0,Y 217.785,Z 520.965,A -85,B 0,C 180,E1 -20720.322,E2 -20720.322} C_VEL
LIN {X 0,Y 215.329,Z 507.307,A -85,B 0,C 180,E1 -20722.153,E2 -20722.153} C_VEL
LIN {X 0,Y 213.103,Z 494.095,A -85,B 0,C 180,E1 -20723.553,E2 -20723.553} C_VEL
LIN {X 0,Y 212.47,Z 490.023,A -85,B 0,C 180,E1 -20723.969,E2 -20723.969} C_VEL
LIN {X 0,Y 212.755,Z 489.986,A -85,B 0,C 180,E1 -20727.547,E2 -20727.547} C_VEL
LIN {X 0,Y 213.206,Z 489.925,A -85,B 0,C 180,E1 -20731.832,E2 -20731.832} C_VEL
LIN {X 0,Y 213.503,Z 489.889,A -85,B 0,C 180,E1 -20734.619,E2 -20734.619} C_VEL
LIN {X 0,Y 213.668,Z 489.868,A -85,B 0,C 180,E1 -20738.679,E2 -20738.679} C_VEL
LIN {X 0,Y 213.707,Z 489.859,A -85,B 0,C 180,E1 -20741.127,E2 -20741.127} C_VEL
LIN {X 0,Y 213.708,Z 489.862,A -85,B 0,C 180,E1 -20743.679,E2 -20743.679} C_VEL
LIN {X 0,Y 213.711,Z 489.865,A -85,B 0,C 180,E1 -20746.344,E2 -20746.344} C_VEL
LIN {X 0,Y 213.74,Z 489.856,A -85,B 0,C 180,E1 -20751.336,E2 -20751.336} C_VEL
LIN {X 0,Y 213.773,Z 489.857,A -85,B 0,C 180,E1 -20756.02,E2 -20756.02} C_VEL
LIN {X 0,Y 213.785,Z 489.854,A -85,B 0,C 180,E1 -20760.454,E2 -20760.454} C_VEL
LIN {X 0,Y 213.806,Z 489.851,A -85,B 0,C 180,E1 -20764.702,E2 -20764.702} C_VEL
LIN {X 0,Y 213.818,Z 489.847,A -85,B 0,C 180,E1 -20768.803,E2 -20768.803} C_VEL
LIN {X 0,Y 213.949,Z 489.833,A -85,B 0,C 180,E1 -20772.804,E2 -20772.804} C_VEL
LIN {X 0,Y 213.958,Z 489.828,A -85,B 0,C 180,E1 -20776.706,E2 -20776.706} C_VEL
LIN {X 0,Y 214.147,Z 489.809,A -85,B 0,C 180,E1 -20780.555,E2 -20780.555} C_VEL
LIN {X 0,Y 214.105,Z 489.812,A -85,B 0,C 180,E1 -20784.348,E2 -20784.348} C_VEL
LIN {X 0,Y 214.45,Z 489.773,A -85,B 0,C 180,E1 -20788.122,E2 -20788.122} C_VEL
LIN {X 0,Y 214.555,Z 489.761,A -85,B 0,C 180,E1 -20790,E2 -20790} C_VEL
LIN {X 0,Y 214.449,Z 489.773,A -85,B 0,C 180,E1 -20791.878,E2 -20791.878} C_VEL
LIN {X 0,Y 214.193,Z 489.803,A -85,B 0,C 180,E1 -20797.541,E2 -20797.541} C_VEL
LIN {X 0,Y 214.012,Z 489.825,A -85,B 0,C 180,E1 -20801.363,E2 -20801.363} C_VEL
LIN {X 0,Y 213.938,Z 489.833,A -85,B 0,C 180,E1 -20805.236,E2 -20805.236} C_VEL
LIN {X 0,Y 213.844,Z 489.846,A -85,B 0,C 180,E1 -20809.187,E2 -20809.187} C_VEL
LIN {X 0,Y 213.851,Z 489.843,A -85,B 0,C 180,E1 -20813.226,E2 -20813.226} C_VEL
LIN {X 0,Y 213.832,Z 489.849,A -85,B 0,C 180,E1 -20817.449,E2 -20817.449} C_VEL
LIN {X 0,Y 213.782,Z 489.853,A -85,B 0,C 180,E1 -20821.735,E2 -20821.735} C_VEL
LIN {X 0,Y 213.755,Z 489.857,A -85,B 0,C 180,E1 -20826.286,E2 -20826.286} C_VEL
LIN {X 0,Y 213.718,Z 489.86,A -85,B 0,C 180,E1 -20831.123,E2 -20831.123} C_VEL
LIN {X 0,Y 213.709,Z 489.866,A -85,B 0,C 180,E1 -20833.677,E2 -20833.677} C_VEL
LIN {X 0,Y 213.707,Z 489.862,A -85,B 0,C 180,E1 -20836.343,E2 -20836.343} C_VEL
LIN {X 0,Y 213.718,Z 489.859,A -85,B 0,C 180,E1 -20839.142,E2 -20839.142} C_VEL
LIN {X 0,Y 213.746,Z 489.861,A -85,B 0,C 180,E1 -20843.711,E2 -20843.711} C_VEL
LIN {X 0,Y 213.797,Z 489.85,A -85,B 0,C 180,E1 -20848.724,E2 -20848.724} C_VEL
LIN {X 0,Y 213.827,Z 489.848,A -85,B 0,C 180,E1 -20852.603,E2 -20852.603} C_VEL
LIN {X 0,Y 213.853,Z 489.842,A -85,B 0,C 180,E1 -20856.952,E2 -20856.952} C_VEL
LIN {X 0,Y 213.945,Z 489.832,A -85,B 0,C 180,E1 -20862.803,E2 -20862.803} C_VEL
LIN {X 0,Y 213.982,Z 489.827,A -85,B 0,C 180,E1 -20866.708,E2 -20866.708} C_VEL
LIN {X 0,Y 214.197,Z 489.801,A -85,B 0,C 180,E1 -20870.557,E2 -20870.557} C_VEL
LIN {X 0,Y 214.249,Z 489.793,A -85,B 0,C 180,E1 -20872.46,E2 -20872.46} C_VEL
LIN {X 0,Y 214.447,Z 489.771,A -85,B 0,C 180,E1 -20878.121,E2 -20878.121} C_VEL
LIN {X 0,Y 214.551,Z 489.757,A -85,B 0,C 180,E1 -20880,E2 -20880} C_VEL
LIN {X 0,Y 214.447,Z 489.768,A -85,B 0,C 180,E1 -20881.878,E2 -20881.878} C_VEL
LIN {X 0,Y 214.248,Z 489.798,A -85,B 0,C 180,E1 -20887.539,E2 -20887.539} C_VEL
LIN {X 0,Y 214.048,Z 489.82,A -85,B 0,C 180,E1 -20891.361,E2 -20891.361} C_VEL
LIN {X 0,Y 213.934,Z 489.837,A -85,B 0,C 180,E1 -20895.236,E2 -20895.236} C_VEL
LIN {X 0,Y 213.868,Z 489.843,A -85,B 0,C 180,E1 -20899.184,E2 -20899.184} C_VEL
LIN {X 0,Y 213.847,Z 489.848,A -85,B 0,C 180,E1 -20903.227,E2 -20903.227} C_VEL
LIN {X 0,Y 213.828,Z 489.847,A -85,B 0,C 180,E1 -20907.45,E2 -20907.45} C_VEL
LIN {X 0,Y 213.769,Z 489.856,A -85,B 0,C 180,E1 -20911.737,E2 -20911.737} C_VEL
LIN {X 0,Y 213.756,Z 489.854,A -85,B 0,C 180,E1 -20916.286,E2 -20916.286} C_VEL
LIN {X 0,Y 213.849,Z 489.847,A -85,B 0,C 180,E1 -20921.093,E2 -20921.093} C_VEL
LIN {X 0,Y 214.042,Z 490.004,A -85,B 0,C 180,E1 -20923.751,E2 -20923.751} C_VEL
LIN {X 0,Y 215.028,Z 495.349,A -85,B 0,C 180,E1 -20929.181,E2 -20929.181} C_VEL
LIN {X 0,Y 215.598,Z 499.173,A -85,B 0,C 180,E1 -20932.911,E2 -20932.911} C_VEL
LIN {X 0,Y 215.365,Z 501.041,A -85,B 0,C 180,E1 -20934.669,E2 -20934.669} C_VEL
LIN {X 0,Y 214.087,Z 506.215,A -85,B 0,C 180,E1 -20939.491,E2 -20939.491} C_VEL
LIN {X 0,Y 212.975,Z 511.686,A -85,B 0,C 180,E1 -20944.597,E2 -20944.597} C_VEL
LIN {X 0,Y 212.79,Z 512.845,A -85,B 0,C 180,E1 -20945.681,E2 -20945.681} C_VEL
LIN {X 0,Y 213.37,Z 527.734,A -85,B 0,C 180,E1 -20947.065,E2 -20947.065} C_VEL
LIN {X 0,Y 214.396,Z 540.711,A -85,B 0,C 180,E1 -20948.633,E2 -20948.633} C_VEL
LIN {X 0,Y 215.641,Z 553.615,A -85,B 0,C 180,E1 -20950.575,E2 -20950.575} C_VEL
LIN {X 0,Y 216.14,Z 560.296,A -85,B 0,C 180,E1 -20951.762,E2 -20951.762} C_VEL
LIN {X 0,Y 214.937,Z 570.324,A -85,B 0,C 180,E1 -20953.864,E2 -20953.864} C_VEL
LIN {X 0,Y 213.983,Z 579.61,A -85,B 0,C 180,E1 -20956.225,E2 -20956.225} C_VEL
LIN {X 0,Y 213.753,Z 581.686,A -85,B 0,C 180,E1 -20956.824,E2 -20956.824} C_VEL
LIN {X 0,Y 213.249,Z 584.267,A -85,B 0,C 180,E1 -20957.61,E2 -20957.61} C_VEL
LIN {X 0,Y 210.956,Z 588.856,A -85,B 0,C 180,E1 -20959.238,E2 -20959.238} C_VEL
LIN {X 0,Y 206.35,Z 595.801,A -85,B 0,C 180,E1 -20962.327,E2 -20962.327} C_VEL
LIN {X 0,Y 205.597,Z 598.649,A -85,B 0,C 180,E1 -20963.761,E2 -20963.761} C_VEL
LIN {X 0,Y 205.561,Z 604.47,A -85,B 0,C 180,E1 -20967.061,E2 -20967.061} C_VEL
LIN {X 0,Y 205.583,Z 608.397,A -85,B 0,C 180,E1 -20970,E2 -20970} C_VEL
LIN {X 0,Y 205.258,Z 610.319,A -85,B 0,C 180,E1 -20971.963,E2 -20971.963} C_VEL
LIN {X 0,Y 204.825,Z 612.961,A -85,B 0,C 180,E1 -20975.909,E2 -20975.909} C_VEL
LIN {X 0,Y 205.115,Z 614.188,A -85,B 0,C 180,E1 -20979.865,E2 -20979.865} C_VEL
LIN {X 0,Y 206.341,Z 614.04,A -85,B 0,C 180,E1 -20983.794,E2 -20983.794} C_VEL
LIN {X 0,Y 208.853,Z 612.607,A -85,B 0,C 180,E1 -20987.63,E2 -20987.63} C_VEL
LIN {X 0,Y 212.412,Z 609.892,A -85,B 0,C 180,E1 -20991.344,E2 -20991.344} C_VEL
LIN {X 0,Y 217.293,Z 605.684,A -85,B 0,C 180,E1 -20995.094,E2 -20995.094} C_VEL
LIN {X 0,Y 222.882,Z 600.593,A -85,B 0,C 180,E1 -20998.229,E2 -20998.229} C_VEL
LIN {X 0,Y 229.775,Z 593.758,A -85,B 0,C 180,E1 -21001.331,E2 -21001.331} C_VEL
LIN {X 0,Y 235.281,Z 587.762,A -85,B 0,C 180,E1 -21003.547,E2 -21003.547} C_VEL
LIN {X 0,Y 237.461,Z 584.698,A -85,B 0,C 180,E1 -21004.732,E2 -21004.732} C_VEL
LIN {X 0,Y 240.751,Z 578.943,A -85,B 0,C 180,E1 -21007.22,E2 -21007.22} C_VEL
LIN {X 0,Y 243.131,Z 574.215,A -85,B 0,C 180,E1 -21009.49,E2 -21009.49} C_VEL
LIN {X 0,Y 244.63,Z 570.914,A -85,B 0,C 180,E1 -21011.359,E2 -21011.359} C_VEL
LIN {X 0,Y 245.465,Z 568.446,A -85,B 0,C 180,E1 -21013.406,E2 -21013.406} C_VEL
LIN {X 0,Y 246.057,Z 566.798,A -85,B 0,C 180,E1 -21015.567,E2 -21015.567} C_VEL
LIN {X 0,Y 246.191,Z 566.383,A -85,B 0,C 180,E1 -21016.755,E2 -21016.755} C_VEL
LIN {X 0,Y 246.048,Z 566.454,A -85,B 0,C 180,E1 -21018.932,E2 -21018.932} C_VEL
LIN {X 0,Y 245.957,Z 567.127,A -85,B 0,C 180,E1 -21021.051,E2 -21021.051} C_VEL
LIN {X 0,Y 245.791,Z 568.45,A -85,B 0,C 180,E1 -21023.19,E2 -21023.19} C_VEL
LIN {X 0,Y 245.354,Z 570.288,A -85,B 0,C 180,E1 -21025.048,E2 -21025.048} C_VEL
LIN {X 0,Y 244.903,Z 571.392,A -85,B 0,C 180,E1 -21025.973,E2 -21025.973} C_VEL
LIN {X 0,Y 243.482,Z 573.206,A -85,B 0,C 180,E1 -21026.741,E2 -21026.741} C_VEL
LIN {X 0,Y 237.509,Z 579.099,A -85,B 0,C 180,E1 -21028.813,E2 -21028.813} C_VEL
LIN {X 0,Y 230.166,Z 585.445,A -85,B 0,C 180,E1 -21031.753,E2 -21031.753} C_VEL
LIN {X 0,Y 223.776,Z 590.23,A -85,B 0,C 180,E1 -21034.914,E2 -21034.914} C_VEL
LIN {X 0,Y 219.557,Z 592.896,A -85,B 0,C 180,E1 -21037.411,E2 -21037.411} C_VEL
LIN {X 0,Y 214.798,Z 595.231,A -85,B 0,C 180,E1 -21040.902,E2 -21040.902} C_VEL
LIN {X 0,Y 210.987,Z 596.228,A -85,B 0,C 180,E1 -21044.545,E2 -21044.545} C_VEL
LIN {X 0,Y 208.048,Z 595.901,A -85,B 0,C 180,E1 -21048.306,E2 -21048.306} C_VEL
LIN {X 0,Y 206.16,Z 594.212,A -85,B 0,C 180,E1 -21052.163,E2 -21052.163} C_VEL
LIN {X 0,Y 205.247,Z 591.081,A -85,B 0,C 180,E1 -21056.074,E2 -21056.074} C_VEL
LIN {X 0,Y 204.766,Z 586.435,A -85,B 0,C 180,E1 -21060,E2 -21060} C_VEL
LIN {X 0,Y 204.806,Z 581.837,A -85,B 0,C 180,E1 -21062.951,E2 -21062.951} C_VEL
LIN {X 0,Y 204.984,Z 575.638,A -85,B 0,C 180,E1 -21066.126,E2 -21066.126} C_VEL
LIN {X 0,Y 205.555,Z 567.767,A -85,B 0,C 180,E1 -21069.347,E2 -21069.347} C_VEL
LIN {X 0,Y 206.429,Z 558.991,A -85,B 0,C 180,E1 -21072.286,E2 -21072.286} C_VEL
LIN {X 0,Y 207.352,Z 550.223,A -85,B 0,C 180,E1 -21074.727,E2 -21074.727} C_VEL
LIN {X 0,Y 208.609,Z 539.707,A -85,B 0,C 180,E1 -21077.145,E2 -21077.145} C_VEL
LIN {X 0,Y 209.843,Z 529.6,A -85,B 0,C 180,E1 -21079.06,E2 -21079.06} C_VEL
LIN {X 0,Y 210.673,Z 521.848,A -85,B 0,C 180,E1 -21080.319,E2 -21080.319} C_VEL
LIN {X 0,Y 208.406,Z 508.827,A -85,B 0,C 180,E1 -21082.145,E2 -21082.145} C_VEL
LIN {X 0,Y 206.248,Z 496.115,A -85,B 0,C 180,E1 -21083.589,E2 -21083.589} C_VEL
LIN {X 0,Y 205.42,Z 490.9,A -85,B 0,C 180,E1 -21084.114,E2 -21084.114} C_VEL
LIN {X 0,Y 205.785,Z 490.852,A -85,B 0,C 180,E1 -21088.564,E2 -21088.564} C_VEL
LIN {X 0,Y 206.273,Z 490.785,A -85,B 0,C 180,E1 -21093.035,E2 -21093.035} C_VEL
LIN {X 0,Y 206.476,Z 490.763,A -85,B 0,C 180,E1 -21095.356,E2 -21095.356} C_VEL
LIN {X 0,Y 206.631,Z 490.746,A -85,B 0,C 180,E1 -21098.529,E2 -21098.529} C_VEL
LIN {X 0,Y 206.625,Z 490.744,A -85,B 0,C 180,E1 -21102.865,E2 -21102.865} C_VEL
LIN {X 0,Y 206.63,Z 490.744,A -85,B 0,C 180,E1 -21107.136,E2 -21107.136} C_VEL
LIN {X 0,Y 206.706,Z 490.732,A -85,B 0,C 180,E1 -21111.445,E2 -21111.445} C_VEL
LIN {X 0,Y 206.735,Z 490.732,A -85,B 0,C 180,E1 -21114.695,E2 -21114.695} C_VEL
LIN {X 0,Y 206.728,Z 490.728,A -85,B 0,C 180,E1 -21119.339,E2 -21119.339} C_VEL
LIN {X 0,Y 206.737,Z 490.733,A -85,B 0,C 180,E1 -21123.772,E2 -21123.772} C_VEL
LIN {X 0,Y 206.763,Z 490.727,A -85,B 0,C 180,E1 -21128.043,E2 -21128.043} C_VEL
LIN {X 0,Y 206.879,Z 490.717,A -85,B 0,C 180,E1 -21132.197,E2 -21132.197} C_VEL
LIN {X 0,Y 206.9,Z 490.709,A -85,B 0,C 180,E1 -21136.244,E2 -21136.244} C_VEL
LIN {X 0,Y 207.104,Z 490.688,A -85,B 0,C 180,E1 -21140.231,E2 -21140.231} C_VEL
LIN {X 0,Y 207.066,Z 490.69,A -85,B 0,C 180,E1 -21144.155,E2 -21144.155} C_VEL
LIN {X 0,Y 207.387,Z 490.652,A -85,B 0,C 180,E1 -21148.058,E2 -21148.058} C_VEL
LIN {X 0,Y 207.52,Z 490.637,A -85,B 0,C 180,E1 -21150,E2 -21150} C_VEL
LIN {X 0,Y 207.385,Z 490.653,A -85,B 0,C 180,E1 -21151.942,E2 -21151.942} C_VEL
LIN {X 0,Y 207.137,Z 490.683,A -85,B 0,C 180,E1 -21157.8,E2 -21157.8} C_VEL
LIN {X 0,Y 206.936,Z 490.708,A -85,B 0,C 180,E1 -21161.757,E2 -21161.757} C_VEL
LIN {X 0,Y 206.872,Z 490.716,A -85,B 0,C 180,E1 -21165.77,E2 -21165.77} C_VEL
LIN {X 0,Y 206.788,Z 490.726,A -85,B 0,C 180,E1 -21169.868,E2 -21169.868} C_VEL
LIN {X 0,Y 206.767,Z 490.729,A -85,B 0,C 180,E1 -21174.071,E2 -21174.071} C_VEL
LIN {X 0,Y 206.747,Z 490.729,A -85,B 0,C 180,E1 -21178.418,E2 -21178.418} C_VEL
LIN {X 0,Y 206.712,Z 490.733,A -85,B 0,C 180,E1 -21182.955,E2 -21182.955} C_VEL
LIN {X 0,Y 206.724,Z 490.734,A -85,B 0,C 180,E1 -21185.32,E2 -21185.32} C_VEL
LIN {X 0,Y 206.668,Z 490.738,A -85,B 0,C 180,E1 -21190.249,E2 -21190.249} C_VEL
LIN {X 0,Y 206.635,Z 490.746,A -85,B 0,C 180,E1 -21195.581,E2 -21195.581} C_VEL
LIN {X 0,Y 206.662,Z 490.741,A -85,B 0,C 180,E1 -21199.748,E2 -21199.748} C_VEL
LIN {X 0,Y 206.7,Z 490.735,A -85,B 0,C 180,E1 -21204.688,E2 -21204.688} C_VEL
LIN {X 0,Y 206.725,Z 490.733,A -85,B 0,C 180,E1 -21209.339,E2 -21209.339} C_VEL
LIN {X 0,Y 206.734,Z 490.732,A -85,B 0,C 180,E1 -21213.772,E2 -21213.772} C_VEL
LIN {X 0,Y 206.759,Z 490.729,A -85,B 0,C 180,E1 -21218.043,E2 -21218.043} C_VEL
LIN {X 0,Y 206.875,Z 490.713,A -85,B 0,C 180,E1 -21222.196,E2 -21222.196} C_VEL
LIN {X 0,Y 206.915,Z 490.708,A -85,B 0,C 180,E1 -21226.245,E2 -21226.245} C_VEL
LIN {X 0,Y 207.133,Z 490.682,A -85,B 0,C 180,E1 -21230.232,E2 -21230.232} C_VEL
LIN {X 0,Y 207.19,Z 490.672,A -85,B 0,C 180,E1 -21232.201,E2 -21232.201} C_VEL
LIN {X 0,Y 207.384,Z 490.651,A -85,B 0,C 180,E1 -21238.057,E2 -21238.057} C_VEL
LIN {X 0,Y 207.516,Z 490.633,A -85,B 0,C 180,E1 -21240,E2 -21240} C_VEL
LIN {X 0,Y 207.383,Z 490.648,A -85,B 0,C 180,E1 -21241.942,E2 -21241.942} C_VEL
LIN {X 0,Y 207.189,Z 490.676,A -85,B 0,C 180,E1 -21247.798,E2 -21247.798} C_VEL
LIN {X 0,Y 206.983,Z 490.7,A -85,B 0,C 180,E1 -21251.755,E2 -21251.755} C_VEL
LIN {X 0,Y 206.867,Z 490.716,A -85,B 0,C 180,E1 -21255.77,E2 -21255.77} C_VEL
LIN {X 0,Y 206.8,Z 490.721,A -85,B 0,C 180,E1 -21259.867,E2 -21259.867} C_VEL
LIN {X 0,Y 206.763,Z 490.728,A -85,B 0,C 180,E1 -21264.072,E2 -21264.072} C_VEL
LIN {X 0,Y 206.736,Z 490.727,A -85,B 0,C 180,E1 -21268.42,E2 -21268.42} C_VEL
LIN {X 0,Y 206.705,Z 490.737,A -85,B 0,C 180,E1 -21272.956,E2 -21272.956} C_VEL
LIN {X 0,Y 206.727,Z 490.731,A -85,B 0,C 180,E1 -21277.73,E2 -21277.73} C_VEL
LIN {X 0,Y 207,Z 490.716,A -85,B 0,C 180,E1 -21283.77,E2 -21283.77} C_VEL
LIN {X 0,Y 207.714,Z 494.823,A -85,B 0,C 180,E1 -21288.105,E2 -21288.105} C_VEL
LIN {X 0,Y 208.286,Z 497.548,A -85,B 0,C 180,E1 -21290.902,E2 -21290.902} C_VEL
LIN {X 0,Y 208.426,Z 500.685,A -85,B 0,C 180,E1 -21294.024,E2 -21294.024} C_VEL
LIN {X 0,Y 207.013,Z 506.212,A -85,B 0,C 180,E1 -21299.387,E2 -21299.387} C_VEL
LIN {X 0,Y 205.854,Z 511.717,A -85,B 0,C 180,E1 -21304.738,E2 -21304.738} C_VEL
LIN {X 0,Y 205.702,Z 512.571,A -85,B 0,C 180,E1 -21305.528,E2 -21305.528} C_VEL
LIN {X 0,Y 206.17,Z 525.565,A -85,B 0,C 180,E1 -21306.734,E2 -21306.734} C_VEL
LIN {X 0,Y 207.122,Z 538.832,A -85,B 0,C 180,E1 -21308.346,E2 -21308.346} C_VEL
LIN {X 0,Y 208.314,Z 551.561,A -85,B 0,C 180,E1 -21310.283,E2 -21310.283} C_VEL
LIN {X 0,Y 209.121,Z 559.065,A -85,B 0,C 180,E1 -21311.635,E2 -21311.635} C_VEL
LIN {X 0,Y 207.794,Z 570.239,A -85,B 0,C 180,E1 -21314.05,E2 -21314.05} C_VEL
LIN {X 0,Y 206.729,Z 580.867,A -85,B 0,C 180,E1 -21316.918,E2 -21316.918} C_VEL
LIN {X 0,Y 206.004,Z 589.165,A -85,B 0,C 180,E1 -21319.683,E2 -21319.683} C_VEL
LIN {X 0,Y 205.671,Z 596.382,A -85,B 0,C 180,E1 -21322.661,E2 -21322.661} C_VEL
LIN {X 0,Y 205.597,Z 598.649,A -85,B 0,C 180,E1 -21323.761,E2 -21323.761} C_VEL
LIN {X 0,Y 204.901,Z 601.302,A -85,B 0,C 180,E1 -21325.221,E2 -21325.221} C_VEL
LIN {X 0,Y 203.318,Z 603.469,A -85,B 0,C 180,E1 -21326.712,E2 -21326.712} C_VEL
LIN {X 0,Y 199.566,Z 606.922,A -85,B 0,C 180,E1 -21329.823,E2 -21329.823} C_VEL
LIN {X 0,Y 198.273,Z 609.002,A -85,B 0,C 180,E1 -21332.024,E2 -21332.024} C_VEL
LIN {X 0,Y 197.805,Z 611.922,A -85,B 0,C 180,E1 -21336.119,E2 -21336.119} C_VEL
LIN {X 0,Y 198.135,Z 613.38,A -85,B 0,C 180,E1 -21340.216,E2 -21340.216} C_VEL
LIN {X 0,Y 199.43,Z 613.546,A -85,B 0,C 180,E1 -21344.282,E2 -21344.282} C_VEL
LIN {X 0,Y 202.1,Z 612.46,A -85,B 0,C 180,E1 -21348.239,E2 -21348.239} C_VEL
LIN {X 0,Y 205.821,Z 610.13,A -85,B 0,C 180,E1 -21352.062,E2 -21352.062} C_VEL
LIN {X 0,Y 210.606,Z 606.526,A -85,B 0,C 180,E1 -21355.71,E2 -21355.71} C_VEL
LIN {X 0,Y 216.722,Z 601.632,A -85,B 0,C 180,E1 -21359.107,E2 -21359.107} C_VEL
LIN {X 0,Y 223.874,Z 595.371,A -85,B 0,C 180,E1 -21362.255,E2 -21362.255} C_VEL
LIN {X 0,Y 229.625,Z 589.721,A -85,B 0,C 180,E1 -21364.488,E2 -21364.488} C_VEL
LIN {X 0,Y 231.267,Z 587.854,A -85,B 0,C 180,E1 -21365.268,E2 -21365.268} C_VEL
LIN {X 0,Y 234.86,Z 582.543,A -85,B 0,C 180,E1 -21367.725,E2 -21367.725} C_VEL
LIN {X 0,Y 238.059,Z 577.245,A -85,B 0,C 180,E1 -21370.503,E2 -21370.503} C_VEL
LIN {X 0,Y 239.252,Z 575.185,A -85,B 0,C 180,E1 -21371.811,E2 -21371.811} C_VEL
LIN {X 0,Y 240.495,Z 572.331,A -85,B 0,C 180,E1 -21374.536,E2 -21374.536} C_VEL
LIN {X 0,Y 240.966,Z 571.151,A -85,B 0,C 180,E1 -21376.816,E2 -21376.816} C_VEL
LIN {X 0,Y 240.662,Z 571.48,A -85,B 0,C 180,E1 -21380.025,E2 -21380.025} C_VEL
LIN {X 0,Y 240.396,Z 572.396,A -85,B 0,C 180,E1 -21382.125,E2 -21382.125} C_VEL
LIN {X 0,Y 239.889,Z 573.867,A -85,B 0,C 180,E1 -21384.131,E2 -21384.131} C_VEL
LIN {X 0,Y 239.401,Z 575.005,A -85,B 0,C 180,E1 -21385.285,E2 -21385.285} C_VEL
LIN {X 0,Y 235.86,Z 578.318,A -85,B 0,C 180,E1 -21386.546,E2 -21386.546} C_VEL
LIN {X 0,Y 227.903,Z 584.961,A -85,B 0,C 180,E1 -21389.415,E2 -21389.415} C_VEL
LIN {X 0,Y 220.768,Z 589.982,A -85,B 0,C 180,E1 -21392.51,E2 -21392.51} C_VEL
LIN {X 0,Y 216.06,Z 592.834,A -85,B 0,C 180,E1 -21394.985,E2 -21394.985} C_VEL
LIN {X 0,Y 210.531,Z 595.445,A -85,B 0,C 180,E1 -21398.457,E2 -21398.457} C_VEL
LIN {X 0,Y 206.013,Z 596.749,A -85,B 0,C 180,E1 -21402.12,E2 -21402.12} C_VEL
LIN {X 0,Y 202.596,Z 596.744,A -85,B 0,C 180,E1 -21405.947,E2 -21405.947} C_VEL
LIN {X 0,Y 199.966,Z 595.381,A -85,B 0,C 180,E1 -21409.879,E2 -21409.879} C_VEL
LIN {X 0,Y 198.593,Z 592.658,A -85,B 0,C 180,E1 -21413.906,E2 -21413.906} C_VEL
LIN {X 0,Y 197.996,Z 589.678,A -85,B 0,C 180,E1 -21416.948,E2 -21416.948} C_VEL
LIN {X 0,Y 197.699,Z 585.803,A -85,B 0,C 180,E1 -21420,E2 -21420} C_VEL
LIN {X 0,Y 197.746,Z 580.928,A -85,B 0,C 180,E1 -21423.056,E2 -21423.056} C_VEL
LIN {X 0,Y 197.951,Z 574.705,A -85,B 0,C 180,E1 -21426.218,E2 -21426.218} C_VEL
LIN {X 0,Y 198.471,Z 567.646,A -85,B 0,C 180,E1 -21429.17,E2 -21429.17} C_VEL
LIN {X 0,Y 199.31,Z 558.752,A -85,B 0,C 180,E1 -21432.215,E2 -21432.215} C_VEL
LIN {X 0,Y 200.518,Z 547.85,A -85,B 0,C 180,E1 -21435.241,E2 -21435.241} C_VEL
LIN {X 0,Y 201.83,Z 536.853,A -85,B 0,C 180,E1 -21437.74,E2 -21437.74} C_VEL
LIN {X 0,Y 202.929,Z 527.689,A -85,B 0,C 180,E1 -21439.472,E2 -21439.472} C_VEL
LIN {X 0,Y 203.506,Z 521.513,A -85,B 0,C 180,E1 -21440.487,E2 -21440.487} C_VEL
LIN {X 0,Y 200.943,Z 507.319,A -85,B 0,C 180,E1 -21442.51,E2 -21442.51} C_VEL
LIN {X 0,Y 198.676,Z 493.454,A -85,B 0,C 180,E1 -21444.051,E2 -21444.051} C_VEL
LIN {X 0,Y 198.397,Z 491.774,A -85,B 0,C 180,E1 -21444.257,E2 -21444.257} C_VEL
LIN {X 0,Y 198.684,Z 491.738,A -85,B 0,C 180,E1 -21447.831,E2 -21447.831} C_VEL
LIN {X 0,Y 199.14,Z 491.677,A -85,B 0,C 180,E1 -21452.112,E2 -21452.112} C_VEL
LIN {X 0,Y 199.446,Z 491.64,A -85,B 0,C 180,E1 -21455.858,E2 -21455.858} C_VEL
LIN {X 0,Y 199.583,Z 491.621,A -85,B 0,C 180,E1 -21459.335,E2 -21459.335} C_VEL
LIN {X 0,Y 199.574,Z 491.622,A -85,B 0,C 180,E1 -21462.309,E2 -21462.309} C_VEL
LIN {X 0,Y 199.584,Z 491.622,A -85,B 0,C 180,E1 -21465.229,E2 -21465.229} C_VEL
LIN {X 0,Y 199.643,Z 491.613,A -85,B 0,C 180,E1 -21470.679,E2 -21470.679} C_VEL
LIN {X 0,Y 199.639,Z 491.616,A -85,B 0,C 180,E1 -21475.718,E2 -21475.718} C_VEL
LIN {X 0,Y 199.708,Z 491.606,A -85,B 0,C 180,E1 -21478.138,E2 -21478.138} C_VEL
LIN {X 0,Y 199.691,Z 491.609,A -85,B 0,C 180,E1 -21482.772,E2 -21482.772} C_VEL
LIN {X 0,Y 199.743,Z 491.599,A -85,B 0,C 180,E1 -21487.229,E2 -21487.229} C_VEL
LIN {X 0,Y 199.801,Z 491.596,A -85,B 0,C 180,E1 -21491.757,E2 -21491.757} C_VEL
LIN {X 0,Y 199.841,Z 491.59,A -85,B 0,C 180,E1 -21495.748,E2 -21495.748} C_VEL
LIN {X 0,Y 200.027,Z 491.569,A -85,B 0,C 180,E1 -21499.881,E2 -21499.881} C_VEL
LIN {X 0,Y 200.028,Z 491.568,A -85,B 0,C 180,E1 -21503.949,E2 -21503.949} C_VEL
LIN {X 0,Y 200.326,Z 491.531,A -85,B 0,C 180,E1 -21507.989,E2 -21507.989} C_VEL
LIN {X 0,Y 200.484,Z 491.514,A -85,B 0,C 180,E1 -21510,E2 -21510} C_VEL
LIN {X 0,Y 200.027,Z 491.566,A -85,B 0,C 180,E1 -21514.029,E2 -21514.029} C_VEL
LIN {X 0,Y 200.087,Z 491.563,A -85,B 0,C 180,E1 -21518.076,E2 -21518.076} C_VEL
LIN {X 0,Y 199.883,Z 491.583,A -85,B 0,C 180,E1 -21522.178,E2 -21522.178} C_VEL
LIN {X 0,Y 199.809,Z 491.595,A -85,B 0,C 180,E1 -21526.343,E2 -21526.343} C_VEL
LIN {X 0,Y 199.704,Z 491.605,A -85,B 0,C 180,E1 -21530.604,E2 -21530.604} C_VEL
LIN {X 0,Y 199.676,Z 491.61,A -85,B 0,C 180,E1 -21534.983,E2 -21534.983} C_VEL
LIN {X 0,Y 199.678,Z 491.611,A -85,B 0,C 180,E1 -21539.521,E2 -21539.521} C_VEL
LIN {X 0,Y 199.667,Z 491.611,A -85,B 0,C 180,E1 -21542.352,E2 -21542.352} C_VEL
LIN {X 0,Y 199.642,Z 491.614,A -85,B 0,C 180,E1 -21546.759,E2 -21546.759} C_VEL
LIN {X 0,Y 199.641,Z 491.613,A -85,B 0,C 180,E1 -21549.32,E2 -21549.32} C_VEL
LIN {X 0,Y 199.582,Z 491.622,A -85,B 0,C 180,E1 -21554.77,E2 -21554.77} C_VEL
LIN {X 0,Y 199.581,Z 491.62,A -85,B 0,C 180,E1 -21558.004,E2 -21558.004} C_VEL
LIN {X 0,Y 199.612,Z 491.618,A -85,B 0,C 180,E1 -21560.767,E2 -21560.767} C_VEL
LIN {X 0,Y 199.616,Z 491.618,A -85,B 0,C 180,E1 -21565.713,E2 -21565.713} C_VEL
LIN {X 0,Y 199.703,Z 491.607,A -85,B 0,C 180,E1 -21568.137,E2 -21568.137} C_VEL
LIN {X 0,Y 199.688,Z 491.609,A -85,B 0,C 180,E1 -21572.771,E2 -21572.771} C_VEL
LIN {X 0,Y 199.739,Z 491.601,A -85,B 0,C 180,E1 -21577.229,E2 -21577.229} C_VEL
LIN {X 0,Y 199.797,Z 491.597,A -85,B 0,C 180,E1 -21581.757,E2 -21581.757} C_VEL
LIN {X 0,Y 199.849,Z 491.589,A -85,B 0,C 180,E1 -21585.749,E2 -21585.749} C_VEL
LIN {X 0,Y 200.076,Z 491.562,A -85,B 0,C 180,E1 -21589.884,E2 -21589.884} C_VEL
LIN {X 0,Y 200.133,Z 491.552,A -85,B 0,C 180,E1 -21591.925,E2 -21591.925} C_VEL
LIN {X 0,Y 200.323,Z 491.531,A -85,B 0,C 180,E1 -21597.989,E2 -21597.989} C_VEL
LIN {X 0,Y 200.48,Z 491.51,A -85,B 0,C 180,E1 -21600,E2 -21600} C_VEL
LIN {X 0,Y 200.033,Z 491.566,A -85,B 0,C 180,E1 -21604.029,E2 -21604.029} C_VEL
LIN {X 0,Y 200.133,Z 491.554,A -85,B 0,C 180,E1 -21608.074,E2 -21608.074} C_VEL
LIN {X 0,Y 199.915,Z 491.579,A -85,B 0,C 180,E1 -21612.176,E2 -21612.176} C_VEL
LIN {X 0,Y 199.806,Z 491.594,A -85,B 0,C 180,E1 -21616.343,E2 -21616.343} C_VEL
LIN {X 0,Y 199.824,Z 491.59,A -85,B 0,C 180,E1 -21618.453,E2 -21618.453} C_VEL
LIN {X 0,Y 199.737,Z 491.604,A -85,B 0,C 180,E1 -21623.817,E2 -21623.817} C_VEL
LIN {X 0,Y 199.707,Z 491.602,A -85,B 0,C 180,E1 -21628.384,E2 -21628.384} C_VEL
LIN {X 0,Y 199.657,Z 491.613,A -85,B 0,C 180,E1 -21632.349,E2 -21632.349} C_VEL
LIN {X 0,Y 199.654,Z 491.612,A -85,B 0,C 180,E1 -21636.756,E2 -21636.756} C_VEL
LIN {X 0,Y 199.793,Z 491.597,A -85,B 0,C 180,E1 -21641.94,E2 -21641.94} C_VEL
LIN {X 0,Y 199.949,Z 491.618,A -85,B 0,C 180,E1 -21644.038,E2 -21644.038} C_VEL
LIN {X 0,Y 200.66,Z 495.504,A -85,B 0,C 180,E1 -21648.282,E2 -21648.282} C_VEL
LIN {X 0,Y 201.208,Z 498.104,A -85,B 0,C 180,E1 -21651.045,E2 -21651.045} C_VEL
LIN {X 0,Y 201.339,Z 500.582,A -85,B 0,C 180,E1 -21653.601,E2 -21653.601} C_VEL
LIN {X 0,Y 200.423,Z 504.245,A -85,B 0,C 180,E1 -21657.307,E2 -21657.307} C_VEL
LIN {X 0,Y 199.329,Z 508.704,A -85,B 0,C 180,E1 -21661.818,E2 -21661.818} C_VEL
LIN {X 0,Y 198.674,Z 512.122,A -85,B 0,C 180,E1 -21665.302,E2 -21665.302} C_VEL
LIN {X 0,Y 199.126,Z 526.427,A -85,B 0,C 180,E1 -21666.712,E2 -21666.712} C_VEL
LIN {X 0,Y 200.206,Z 541.13,A -85,B 0,C 180,E1 -21668.642,E2 -21668.642} C_VEL
LIN {X 0,Y 201.43,Z 553.501,A -85,B 0,C 180,E1 -21670.687,E2 -21670.687} C_VEL
LIN {X 0,Y 201.993,Z 559.079,A -85,B 0,C 180,E1 -21671.752,E2 -21671.752} C_VEL
LIN {X 0,Y 200.668,Z 570.076,A -85,B 0,C 180,E1 -21674.251,E2 -21674.251} C_VEL
LIN {X 0,Y 199.656,Z 580.756,A -85,B 0,C 180,E1 -21677.291,E2 -21677.291} C_VEL
LIN {X 0,Y 198.958,Z 589.404,A -85,B 0,C 180,E1 -21680.341,E2 -21680.341} C_VEL
LIN {X 0,Y 198.661,Z 596.368,A -85,B 0,C 180,E1 -21683.384,E2 -21683.384} C_VEL
LIN {X 0,Y 198.595,Z 602.821,A -85,B 0,C 180,E1 -21686.958,E2 -21686.958} C_VEL
LIN {X 0,Y 198.618,Z 606.926,A -85,B 0,C 180,E1 -21690,E2 -21690} C_VEL
LIN {X 0,Y 198.273,Z 609.002,A -85,B 0,C 180,E1 -21692.024,E2 -21692.024} C_VEL
LIN {X 0,Y 197.826,Z 609.958,A -85,B 0,C 180,E1 -21693.119,E2 -21693.119} C_VEL
LIN {X 0,Y 196.316,Z 610.999,A -85,B 0,C 180,E1 -21694.757,E2 -21694.757} C_VEL
LIN {X 0,Y 192.001,Z 612.21,A -85,B 0,C 180,E1 -21698.663,E2 -21698.663} C_VEL
LIN {X 0,Y 191.219,Z 612.514,A -85,B 0,C 180,E1 -21700.427,E2 -21700.427} C_VEL
LIN {X 0,Y 191.269,Z 612.619,A -85,B 0,C 180,E1 -21701.021,E2 -21701.021} C_VEL
LIN {X 0,Y 192.541,Z 612.999,A -85,B 0,C 180,E1 -21704.804,E2 -21704.804} C_VEL
LIN {X 0,Y 195.355,Z 612.228,A -85,B 0,C 180,E1 -21708.892,E2 -21708.892} C_VEL
LIN {X 0,Y 199.268,Z 610.232,A -85,B 0,C 180,E1 -21712.828,E2 -21712.828} C_VEL
LIN {X 0,Y 204.262,Z 607.052,A -85,B 0,C 180,E1 -21716.57,E2 -21716.57} C_VEL
LIN {X 0,Y 210.613,Z 602.607,A -85,B 0,C 180,E1 -21720.036,E2 -21720.036} C_VEL
LIN {X 0,Y 218.017,Z 596.856,A -85,B 0,C 180,E1 -21723.231,E2 -21723.231} C_VEL
LIN {X 0,Y 224.007,Z 591.674,A -85,B 0,C 180,E1 -21725.481,E2 -21725.481} C_VEL
LIN {X 0,Y 225.747,Z 589.899,A -85,B 0,C 180,E1 -21726.265,E2 -21726.265} C_VEL
LIN {X 0,Y 229.698,Z 584.885,A -85,B 0,C 180,E1 -21728.847,E2 -21728.847} C_VEL
LIN {X 0,Y 233.019,Z 580.218,A -85,B 0,C 180,E1 -21731.571,E2 -21731.571} C_VEL
LIN {X 0,Y 233.892,Z 578.879,A -85,B 0,C 180,E1 -21732.539,E2 -21732.539} C_VEL
LIN {X 0,Y 234.627,Z 577.407,A -85,B 0,C 180,E1 -21734.037,E2 -21734.037} C_VEL
LIN {X 0,Y 235.295,Z 576.099,A -85,B 0,C 180,E1 -21735.796,E2 -21735.796} C_VEL
LIN {X 0,Y 235.467,Z 575.769,A -85,B 0,C 180,E1 -21736.648,E2 -21736.648} C_VEL
LIN {X 0,Y 235.261,Z 575.715,A -85,B 0,C 180,E1 -21738.913,E2 -21738.913} C_VEL
LIN {X 0,Y 234.865,Z 576.315,A -85,B 0,C 180,E1 -21741.08,E2 -21741.08} C_VEL
LIN {X 0,Y 233.951,Z 578.173,A -85,B 0,C 180,E1 -21744.204,E2 -21744.204} C_VEL
LIN {X 0,Y 232.515,Z 579.548,A -85,B 0,C 180,E1 -21744.95,E2 -21744.95} C_VEL
LIN {X 0,Y 224.093,Z 585.948,A -85,B 0,C 180,E1 -21747.781,E2 -21747.781} C_VEL
LIN {X 0,Y 216.445,Z 590.886,A -85,B 0,C 180,E1 -21750.853,E2 -21750.853} C_VEL
LIN {X 0,Y 209.8,Z 594.403,A -85,B 0,C 180,E1 -21754.184,E2 -21754.184} C_VEL
LIN {X 0,Y 204.041,Z 596.598,A -85,B 0,C 180,E1 -21757.736,E2 -21757.736} C_VEL
LIN {X 0,Y 199.323,Z 597.509,A -85,B 0,C 180,E1 -21761.499,E2 -21761.499} C_VEL
LIN {X 0,Y 195.726,Z 597.131,A -85,B 0,C 180,E1 -21765.443,E2 -21765.443} C_VEL
LIN {X 0,Y 192.984,Z 595.46,A -85,B 0,C 180,E1 -21769.509,E2 -21769.509} C_VEL
LIN {X 0,Y 191.549,Z 592.414,A -85,B 0,C 180,E1 -21773.681,E2 -21773.681} C_VEL
LIN {X 0,Y 190.94,Z 589.194,A -85,B 0,C 180,E1 -21776.836,E2 -21776.836} C_VEL
LIN {X 0,Y 190.621,Z 583.474,A -85,B 0,C 180,E1 -21781.057,E2 -21781.057} C_VEL
LIN {X 0,Y 190.719,Z 577.961,A -85,B 0,C 180,E1 -21784.227,E2 -21784.227} C_VEL
LIN {X 0,Y 191.203,Z 570.012,A -85,B 0,C 180,E1 -21787.923,E2 -21787.923} C_VEL
LIN {X 0,Y 191.908,Z 561.583,A -85,B 0,C 180,E1 -21791.086,E2 -21791.086} C_VEL
LIN {X 0,Y 192.774,Z 553.224,A -85,B 0,C 180,E1 -21793.709,E2 -21793.709} C_VEL
LIN {X 0,Y 194.149,Z 542.155,A -85,B 0,C 180,E1 -21796.564,E2 -21796.564} C_VEL
LIN {X 0,Y 195.645,Z 529.748,A -85,B 0,C 180,E1 -21799.135,E2 -21799.135} C_VEL
LIN {X 0,Y 196.383,Z 522.391,A -85,B 0,C 180,E1 -21800.422,E2 -21800.422} C_VEL
LIN {X 0,Y 194.152,Z 509.614,A -85,B 0,C 180,E1 -21802.34,E2 -21802.34} C_VEL
LIN {X 0,Y 192.102,Z 497.306,A -85,B 0,C 180,E1 -21803.847,E2 -21803.847} C_VEL
LIN {X 0,Y 191.347,Z 492.651,A -85,B 0,C 180,E1 -21804.349,E2 -21804.349} C_VEL
LIN {X 0,Y 191.673,Z 492.61,A -85,B 0,C 180,E1 -21808.469,E2 -21808.469} C_VEL
LIN {X 0,Y 192.155,Z 492.543,A -85,B 0,C 180,E1 -21813.273,E2 -21813.273} C_VEL
LIN {X 0,Y 192.415,Z 492.517,A -85,B 0,C 180,E1 -21816.528,E2 -21816.528} C_VEL
LIN {X 0,Y 192.507,Z 492.5,A -85,B 0,C 180,E1 -21821.083,E2 -21821.083} C_VEL
LIN {X 0,Y 192.517,Z 492.505,A -85,B 0,C 180,E1 -21826.083,E2 -21826.083} C_VEL
LIN {X 0,Y 192.545,Z 492.498,A -85,B 0,C 180,E1 -21830.043,E2 -21830.043} C_VEL
LIN {X 0,Y 192.603,Z 492.495,A -85,B 0,C 180,E1 -21834.279,E2 -21834.279} C_VEL
LIN {X 0,Y 192.612,Z 492.486,A -85,B 0,C 180,E1 -21839.28,E2 -21839.28} C_VEL
LIN {X 0,Y 192.669,Z 492.483,A -85,B 0,C 180,E1 -21841.692,E2 -21841.692} C_VEL
LIN {X 0,Y 192.711,Z 492.478,A -85,B 0,C 180,E1 -21846.349,E2 -21846.349} C_VEL
LIN {X 0,Y 192.737,Z 492.475,A -85,B 0,C 180,E1 -21851.457,E2 -21851.457} C_VEL
LIN {X 0,Y 192.769,Z 492.469,A -85,B 0,C 180,E1 -21855.214,E2 -21855.214} C_VEL
LIN {X 0,Y 192.949,Z 492.449,A -85,B 0,C 180,E1 -21859.566,E2 -21859.566} C_VEL
LIN {X 0,Y 192.99,Z 492.445,A -85,B 0,C 180,E1 -21863.727,E2 -21863.727} C_VEL
LIN {X 0,Y 193.268,Z 492.41,A -85,B 0,C 180,E1 -21867.916,E2 -21867.916} C_VEL
LIN {X 0,Y 193.448,Z 492.39,A -85,B 0,C 180,E1 -21870,E2 -21870} C_VEL
LIN {X 0,Y 192.972,Z 492.444,A -85,B 0,C 180,E1 -21874.177,E2 -21874.177} C_VEL
LIN {X 0,Y 193.035,Z 492.439,A -85,B 0,C 180,E1 -21878.373,E2 -21878.373} C_VEL
LIN {X 0,Y 192.809,Z 492.462,A -85,B 0,C 180,E1 -21882.632,E2 -21882.632} C_VEL
LIN {X 0,Y 192.762,Z 492.472,A -85,B 0,C 180,E1 -21886.958,E2 -21886.958} C_VEL
LIN {X 0,Y 192.641,Z 492.485,A -85,B 0,C 180,E1 -21891.396,E2 -21891.396} C_VEL
LIN {X 0,Y 192.668,Z 492.485,A -85,B 0,C 180,E1 -21894.224,E2 -21894.224} C_VEL
LIN {X 0,Y 192.653,Z 492.484,A -85,B 0,C 180,E1 -21898.891,E2 -21898.891} C_VEL
LIN {X 0,Y 192.603,Z 492.491,A -85,B 0,C 180,E1 -21903.184,E2 -21903.184} C_VEL
LIN {X 0,Y 192.612,Z 492.49,A -85,B 0,C 180,E1 -21906.607,E2 -21906.607} C_VEL
LIN {X 0,Y 192.526,Z 492.499,A -85,B 0,C 180,E1 -21911.077,E2 -21911.077} C_VEL
LIN {X 0,Y 192.493,Z 492.505,A -85,B 0,C 180,E1 -21916.076,E2 -21916.076} C_VEL
LIN {X 0,Y 192.52,Z 492.503,A -85,B 0,C 180,E1 -21920.05,E2 -21920.05} C_VEL
LIN {X 0,Y 192.562,Z 492.497,A -85,B 0,C 180,E1 -21924.27,E2 -21924.27} C_VEL
LIN {X 0,Y 192.612,Z 492.487,A -85,B 0,C 180,E1 -21927.057,E2 -21927.057} C_VEL
LIN {X 0,Y 192.666,Z 492.487,A -85,B 0,C 180,E1 -21931.691,E2 -21931.691} C_VEL
LIN {X 0,Y 192.707,Z 492.476,A -85,B 0,C 180,E1 -21936.348,E2 -21936.348} C_VEL
LIN {X 0,Y 192.733,Z 492.478,A -85,B 0,C 180,E1 -21941.457,E2 -21941.457} C_VEL
LIN {X 0,Y 192.773,Z 492.467,A -85,B 0,C 180,E1 -21945.214,E2 -21945.214} C_VEL
LIN {X 0,Y 193.021,Z 492.443,A -85,B 0,C 180,E1 -21949.51,E2 -21949.51} C_VEL
LIN {X 0,Y 193.006,Z 492.44,A -85,B 0,C 180,E1 -21953.728,E2 -21953.728} C_VEL
LIN {X 0,Y 193.265,Z 492.411,A -85,B 0,C 180,E1 -21957.915,E2 -21957.915} C_VEL
LIN {X 0,Y 193.444,Z 492.386,A -85,B 0,C 180,E1 -21960,E2 -21960} C_VEL
LIN {X 0,Y 192.98,Z 492.444,A -85,B 0,C 180,E1 -21964.176,E2 -21964.176} C_VEL
LIN {X 0,Y 193.08,Z 492.432,A -85,B 0,C 180,E1 -21968.371,E2 -21968.371} C_VEL
LIN {X 0,Y 192.854,Z 492.459,A -85,B 0,C 180,E1 -21972.629,E2 -21972.629} C_VEL
LIN {X 0,Y 192.781,Z 492.467,A -85,B 0,C 180,E1 -21978.586,E2 -21978.586} C_VEL
LIN {X 0,Y 192.664,Z 492.484,A -85,B 0,C 180,E1 -21984.225,E2 -21984.225} C_VEL
LIN {X 0,Y 192.643,Z 492.483,A -85,B 0,C 180,E1 -21988.889,E2 -21988.889} C_VEL
LIN {X 0,Y 192.597,Z 492.495,A -85,B 0,C 180,E1 -21993.186,E2 -21993.186} C_VEL
LIN {X 0,Y 192.613,Z 492.488,A -85,B 0,C 180,E1 -21998.337,E2 -21998.337} C_VEL
LIN {X 0,Y 192.938,Z 492.458,A -85,B 0,C 180,E1 -22004.25,E2 -22004.25} C_VEL
LIN {X 0,Y 193.836,Z 497.162,A -85,B 0,C 180,E1 -22009.588,E2 -22009.588} C_VEL
LIN {X 0,Y 194.263,Z 500.058,A -85,B 0,C 180,E1 -22012.741,E2 -22012.741} C_VEL
LIN {X 0,Y 194.044,Z 501.794,A -85,B 0,C 180,E1 -22014.585,E2 -22014.585} C_VEL
LIN {X 0,Y 192.812,Z 506.277,A -85,B 0,C 180,E1 -22019.317,E2 -22019.317} C_VEL
LIN {X 0,Y 191.59,Z 511.752,A -85,B 0,C 180,E1 -22025.122,E2 -22025.122} C_VEL
LIN {X 0,Y 192.046,Z 526.664,A -85,B 0,C 180,E1 -22026.688,E2 -22026.688} C_VEL
LIN {X 0,Y 193.097,Z 540.975,A -85,B 0,C 180,E1 -22028.657,E2 -22028.657} C_VEL
LIN {X 0,Y 194.319,Z 553.232,A -85,B 0,C 180,E1 -22030.769,E2 -22030.769} C_VEL
LIN {X 0,Y 194.914,Z 558.827,A -85,B 0,C 180,E1 -22031.881,E2 -22031.881} C_VEL
LIN {X 0,Y 193.69,Z 568.696,A -85,B 0,C 180,E1 -22034.209,E2 -22034.209} C_VEL
LIN {X 0,Y 192.789,Z 577.917,A -85,B 0,C 180,E1 -22036.831,E2 -22036.831} C_VEL
LIN {X 0,Y 192.049,Z 586.962,A -85,B 0,C 180,E1 -22039.991,E2 -22039.991} C_VEL
LIN {X 0,Y 191.738,Z 594.154,A -85,B 0,C 180,E1 -22043.085,E2 -22043.085} C_VEL
LIN {X 0,Y 191.625,Z 599.244,A -85,B 0,C 180,E1 -22045.794,E2 -22045.794} C_VEL
LIN {X 0,Y 191.669,Z 604.034,A -85,B 0,C 180,E1 -22048.95,E2 -22048.95} C_VEL
LIN {X 0,Y 191.486,Z 606.546,A -85,B 0,C 180,E1 -22051.052,E2 -22051.052} C_VEL
LIN {X 0,Y 190.955,Z 609.36,A -85,B 0,C 180,E1 -22054.222,E2 -22054.222} C_VEL
LIN {X 0,Y 190.871,Z 611.811,A -85,B 0,C 180,E1 -22058.47,E2 -22058.47} C_VEL
LIN {X 0,Y 191.269,Z 612.619,A -85,B 0,C 180,E1 -22061.021,E2 -22061.021} C_VEL
LIN {X 0,Y 191.136,Z 612.86,A -85,B 0,C 180,E1 -22062.79,E2 -22062.79} C_VEL
LIN {X 0,Y 189.582,Z 612.699,A -85,B 0,C 180,E1 -22065.738,E2 -22065.738} C_VEL
LIN {X 0,Y 188.63,Z 612.125,A -85,B 0,C 180,E1 -22068.718,E2 -22068.718} C_VEL
LIN {X 0,Y 189.427,Z 611.606,A -85,B 0,C 180,E1 -22070.481,E2 -22070.481} C_VEL
LIN {X 0,Y 192.734,Z 610.275,A -85,B 0,C 180,E1 -22073.648,E2 -22073.648} C_VEL
LIN {X 0,Y 197.959,Z 607.483,A -85,B 0,C 180,E1 -22077.486,E2 -22077.486} C_VEL
LIN {X 0,Y 204.561,Z 603.516,A -85,B 0,C 180,E1 -22081.021,E2 -22081.021} C_VEL
LIN {X 0,Y 212.2,Z 598.257,A -85,B 0,C 180,E1 -22084.266,E2 -22084.266} C_VEL
LIN {X 0,Y 218.425,Z 593.47,A -85,B 0,C 180,E1 -22086.531,E2 -22086.531} C_VEL
LIN {X 0,Y 220.25,Z 591.82,A -85,B 0,C 180,E1 -22087.321,E2 -22087.321} C_VEL
LIN {X 0,Y 223.13,Z 588.758,A -85,B 0,C 180,E1 -22089.047,E2 -22089.047} C_VEL
LIN {X 0,Y 225.676,Z 585.795,A -85,B 0,C 180,E1 -22090.843,E2 -22090.843} C_VEL
LIN {X 0,Y 227.889,Z 583.042,A -85,B 0,C 180,E1 -22092.725,E2 -22092.725} C_VEL
LIN {X 0,Y 229.289,Z 580.893,A -85,B 0,C 180,E1 -22095.172,E2 -22095.172} C_VEL
LIN {X 0,Y 229.703,Z 579.969,A -85,B 0,C 180,E1 -22097.692,E2 -22097.692} C_VEL
LIN {X 0,Y 229.276,Z 580.211,A -85,B 0,C 180,E1 -22100.026,E2 -22100.026} C_VEL
LIN {X 0,Y 228.385,Z 581.489,A -85,B 0,C 180,E1 -22103.139,E2 -22103.139} C_VEL
LIN {X 0,Y 227.119,Z 582.544,A -85,B 0,C 180,E1 -22103.989,E2 -22103.989} C_VEL
LIN {X 0,Y 218.403,Z 588.421,A -85,B 0,C 180,E1 -22106.836,E2 -22106.836} C_VEL
LIN {X 0,Y 210.492,Z 592.803,A -85,B 0,C 180,E1 -22109.946,E2 -22109.946} C_VEL
LIN {X 0,Y 203.562,Z 595.856,A -85,B 0,C 180,E1 -22113.332,E2 -22113.332} C_VEL
LIN {X 0,Y 197.564,Z 597.664,A -85,B 0,C 180,E1 -22116.965,E2 -22116.965} C_VEL
LIN {X 0,Y 192.662,Z 598.199,A -85,B 0,C 180,E1 -22120.834,E2 -22120.834} C_VEL
LIN {X 0,Y 188.881,Z 597.443,A -85,B 0,C 180,E1 -22124.903,E2 -22124.903} C_VEL
LIN {X 0,Y 186.021,Z 595.402,A -85,B 0,C 180,E1 -22129.112,E2 -22129.112} C_VEL
LIN {X 0,Y 184.51,Z 592.044,A -85,B 0,C 180,E1 -22133.439,E2 -22133.439} C_VEL
LIN {X 0,Y 183.887,Z 588.575,A -85,B 0,C 180,E1 -22136.714,E2 -22136.714} C_VEL
LIN {X 0,Y 183.589,Z 582.514,A -85,B 0,C 180,E1 -22141.097,E2 -22141.097} C_VEL
LIN {X 0,Y 183.728,Z 575.428,A -85,B 0,C 180,E1 -22145.051,E2 -22145.051} C_VEL
LIN {X 0,Y 184.227,Z 568.394,A -85,B 0,C 180,E1 -22148.225,E2 -22148.225} C_VEL
LIN {X 0,Y 184.979,Z 559.581,A -85,B 0,C 180,E1 -22151.506,E2 -22151.506} C_VEL
LIN {X 0,Y 186.151,Z 548.826,A -85,B 0,C 180,E1 -22154.765,E2 -22154.765} C_VEL
LIN {X 0,Y 187.412,Z 538.008,A -85,B 0,C 180,E1 -22157.458,E2 -22157.458} C_VEL
LIN {X 0,Y 188.745,Z 527.599,A -85,B 0,C 180,E1 -22159.58,E2 -22159.58} C_VEL
LIN {X 0,Y 189.239,Z 522.448,A -85,B 0,C 180,E1 -22160.488,E2 -22160.488} C_VEL
LIN {X 0,Y 186.808,Z 508.824,A -85,B 0,C 180,E1 -22162.597,E2 -22162.597} C_VEL
LIN {X 0,Y 184.392,Z 494,A -85,B 0,C 180,E1 -22164.397,E2 -22164.397} C_VEL
LIN {X 0,Y 184.341,Z 493.523,A -85,B 0,C 180,E1 -22164.532,E2 -22164.532} C_VEL
LIN {X 0,Y 184.708,Z 493.476,A -85,B 0,C 180,E1 -22169.647,E2 -22169.647} C_VEL
LIN {X 0,Y 185.112,Z 493.421,A -85,B 0,C 180,E1 -22173.356,E2 -22173.356} C_VEL
LIN {X 0,Y 185.37,Z 493.393,A -85,B 0,C 180,E1 -22177.346,E2 -22177.346} C_VEL
LIN {X 0,Y 185.46,Z 493.378,A -85,B 0,C 180,E1 -22180.72,E2 -22180.72} C_VEL
LIN {X 0,Y 185.483,Z 493.381,A -85,B 0,C 180,E1 -22186.049,E2 -22186.049} C_VEL
LIN {X 0,Y 185.493,Z 493.376,A -85,B 0,C 180,E1 -22189.901,E2 -22189.901} C_VEL
LIN {X 0,Y 185.548,Z 493.371,A -85,B 0,C 180,E1 -22192.696,E2 -22192.696} C_VEL
LIN {X 0,Y 185.549,Z 493.371,A -85,B 0,C 180,E1 -22197.975,E2 -22197.975} C_VEL
LIN {X 0,Y 185.586,Z 493.366,A -85,B 0,C 180,E1 -22200.576,E2 -22200.576} C_VEL
LIN {X 0,Y 185.592,Z 493.365,A -85,B 0,C 180,E1 -22205.383,E2 -22205.383} C_VEL
LIN {X 0,Y 185.612,Z 493.363,A -85,B 0,C 180,E1 -22210.075,E2 -22210.075} C_VEL
LIN {X 0,Y 185.7,Z 493.351,A -85,B 0,C 180,E1 -22214.637,E2 -22214.637} C_VEL
LIN {X 0,Y 185.893,Z 493.327,A -85,B 0,C 180,E1 -22219.417,E2 -22219.417} C_VEL
LIN {X 0,Y 185.953,Z 493.32,A -85,B 0,C 180,E1 -22223.489,E2 -22223.489} C_VEL
LIN {X 0,Y 186.212,Z 493.288,A -85,B 0,C 180,E1 -22227.837,E2 -22227.837} C_VEL
LIN {X 0,Y 186.411,Z 493.266,A -85,B 0,C 180,E1 -22230,E2 -22230} C_VEL
LIN {X 0,Y 185.919,Z 493.322,A -85,B 0,C 180,E1 -22234.335,E2 -22234.335} C_VEL
LIN {X 0,Y 185.983,Z 493.317,A -85,B 0,C 180,E1 -22238.693,E2 -22238.693} C_VEL
LIN {X 0,Y 185.735,Z 493.343,A -85,B 0,C 180,E1 -22243.122,E2 -22243.122} C_VEL
LIN {X 0,Y 185.694,Z 493.354,A -85,B 0,C 180,E1 -22247.624,E2 -22247.624} C_VEL
LIN {X 0,Y 185.601,Z 493.362,A -85,B 0,C 180,E1 -22252.25,E2 -22252.25} C_VEL
LIN {X 0,Y 185.566,Z 493.369,A -85,B 0,C 180,E1 -22257.031,E2 -22257.031} C_VEL
LIN {X 0,Y 185.582,Z 493.366,A -85,B 0,C 180,E1 -22259.492,E2 -22259.492} C_VEL
LIN {X 0,Y 185.522,Z 493.374,A -85,B 0,C 180,E1 -22264.627,E2 -22264.627} C_VEL
LIN {X 0,Y 185.546,Z 493.371,A -85,B 0,C 180,E1 -22267.303,E2 -22267.303} C_VEL
LIN {X 0,Y 185.487,Z 493.376,A -85,B 0,C 180,E1 -22270.729,E2 -22270.729} C_VEL
LIN {X 0,Y 185.462,Z 493.381,A -85,B 0,C 180,E1 -22276.054,E2 -22276.054} C_VEL
LIN {X 0,Y 185.47,Z 493.381,A -85,B 0,C 180,E1 -22279.895,E2 -22279.895} C_VEL
LIN {X 0,Y 185.508,Z 493.376,A -85,B 0,C 180,E1 -22282.71,E2 -22282.71} C_VEL
LIN {X 0,Y 185.548,Z 493.37,A -85,B 0,C 180,E1 -22287.975,E2 -22287.975} C_VEL
LIN {X 0,Y 185.583,Z 493.366,A -85,B 0,C 180,E1 -22290.575,E2 -22290.575} C_VEL
LIN {X 0,Y 185.589,Z 493.364,A -85,B 0,C 180,E1 -22295.382,E2 -22295.382} C_VEL
LIN {X 0,Y 185.676,Z 493.356,A -85,B 0,C 180,E1 -22301.132,E2 -22301.132} C_VEL
LIN {X 0,Y 185.766,Z 493.342,A -85,B 0,C 180,E1 -22306.879,E2 -22306.879} C_VEL
LIN {X 0,Y 186.03,Z 493.312,A -85,B 0,C 180,E1 -22311.308,E2 -22311.308} C_VEL
LIN {X 0,Y 186.209,Z 493.29,A -85,B 0,C 180,E1 -22317.836,E2 -22317.836} C_VEL
LIN {X 0,Y 186.408,Z 493.263,A -85,B 0,C 180,E1 -22319.999,E2 -22319.999} C_VEL
LIN {X 0,Y 185.928,Z 493.322,A -85,B 0,C 180,E1 -22324.335,E2 -22324.335} C_VEL
LIN {X 0,Y 186.029,Z 493.31,A -85,B 0,C 180,E1 -22328.691,E2 -22328.691} C_VEL
LIN {X 0,Y 185.765,Z 493.343,A -85,B 0,C 180,E1 -22333.12,E2 -22333.12} C_VEL
LIN {X 0,Y 185.717,Z 493.349,A -85,B 0,C 180,E1 -22337.622,E2 -22337.622} C_VEL
LIN {X 0,Y 185.6,Z 493.364,A -85,B 0,C 180,E1 -22342.251,E2 -22342.251} C_VEL
LIN {X 0,Y 185.56,Z 493.37,A -85,B 0,C 180,E1 -22347.032,E2 -22347.032} C_VEL
LIN {X 0,Y 185.577,Z 493.366,A -85,B 0,C 180,E1 -22349.493,E2 -22349.493} C_VEL
LIN {X 0,Y 185.52,Z 493.374,A -85,B 0,C 180,E1 -22354.627,E2 -22354.627} C_VEL
LIN {X 0,Y 185.567,Z 493.366,A -85,B 0,C 180,E1 -22357.314,E2 -22357.314} C_VEL
LIN {X 0,Y 185.788,Z 493.342,A -85,B 0,C 180,E1 -22362.914,E2 -22362.914} C_VEL
LIN {X 0,Y 185.954,Z 493.52,A -85,B 0,C 180,E1 -22364.877,E2 -22364.877} C_VEL
LIN {X 0,Y 186.875,Z 498.15,A -85,B 0,C 180,E1 -22370.258,E2 -22370.258} C_VEL
LIN {X 0,Y 187.125,Z 500.628,A -85,B 0,C 180,E1 -22373.064,E2 -22373.064} C_VEL
LIN {X 0,Y 186.523,Z 503.288,A -85,B 0,C 180,E1 -22375.989,E2 -22375.989} C_VEL
LIN {X 0,Y 185.342,Z 507.56,A -85,B 0,C 180,E1 -22380.708,E2 -22380.708} C_VEL
LIN {X 0,Y 184.515,Z 511.555,A -85,B 0,C 180,E1 -22385.005,E2 -22385.005} C_VEL
LIN {X 0,Y 184.839,Z 524.75,A -85,B 0,C 180,E1 -22386.407,E2 -22386.407} C_VEL
LIN {X 0,Y 185.741,Z 538.053,A -85,B 0,C 180,E1 -22388.25,E2 -22388.25} C_VEL
LIN {X 0,Y 187.037,Z 551.558,A -85,B 0,C 180,E1 -22390.592,E2 -22390.592} C_VEL
LIN {X 0,Y 187.808,Z 558.5,A -85,B 0,C 180,E1 -22392.018,E2 -22392.018} C_VEL
LIN {X 0,Y 186.511,Z 569.35,A -85,B 0,C 180,E1 -22394.707,E2 -22394.707} C_VEL
LIN {X 0,Y 185.684,Z 578.3,A -85,B 0,C 180,E1 -22397.43,E2 -22397.43} C_VEL
LIN {X 0,Y 184.986,Z 587.878,A -85,B 0,C 180,E1 -22401.037,E2 -22401.037} C_VEL
LIN {X 0,Y 184.778,Z 595.278,A -85,B 0,C 180,E1 -22404.544,E2 -22404.544} C_VEL
LIN {X 0,Y 184.73,Z 600.768,A -85,B 0,C 180,E1 -22407.82,E2 -22407.82} C_VEL
LIN {X 0,Y 184.753,Z 603.733,A -85,B 0,C 180,E1 -22410,E2 -22410} C_VEL
LIN {X 0,Y 184.393,Z 606.084,A -85,B 0,C 180,E1 -22412.185,E2 -22412.185} C_VEL
LIN {X 0,Y 183.851,Z 609.539,A -85,B 0,C 180,E1 -22416.586,E2 -22416.586} C_VEL
LIN {X 0,Y 184.268,Z 611.601,A -85,B 0,C 180,E1 -22421.199,E2 -22421.199} C_VEL
LIN {X 0,Y 185.683,Z 612.318,A -85,B 0,C 180,E1 -22425.364,E2 -22425.364} C_VEL
LIN {X 0,Y 188.641,Z 611.894,A -85,B 0,C 180,E1 -22429.591,E2 -22429.591} C_VEL
LIN {X 0,Y 189.427,Z 611.606,A -85,B 0,C 180,E1 -22430.481,E2 -22430.481} C_VEL
LIN {X 0,Y 190.44,Z 611.012,A -85,B 0,C 180,E1 -22432.228,E2 -22432.228} C_VEL
LIN {X 0,Y 191.478,Z 608.4,A -85,B 0,C 180,E1 -22437.514,E2 -22437.514} C_VEL
LIN {X 0,Y 193.018,Z 607.233,A -85,B 0,C 180,E1 -22439.167,E2 -22439.167} C_VEL
LIN {X 0,Y 193.833,Z 606.779,A -85,B 0,C 180,E1 -22439.679,E2 -22439.679} C_VEL
LIN {X 0,Y 200.464,Z 603.206,A -85,B 0,C 180,E1 -22442.917,E2 -22442.917} C_VEL
LIN {X 0,Y 208.583,Z 598.141,A -85,B 0,C 180,E1 -22446.133,E2 -22446.133} C_VEL
LIN {X 0,Y 212.916,Z 595.187,A -85,B 0,C 180,E1 -22447.637,E2 -22447.637} C_VEL
LIN {X 0,Y 214.825,Z 593.664,A -85,B 0,C 180,E1 -22448.433,E2 -22448.433} C_VEL
LIN {X 0,Y 219.186,Z 589.501,A -85,B 0,C 180,E1 -22451.096,E2 -22451.096} C_VEL
LIN {X 0,Y 222.075,Z 586.484,A -85,B 0,C 180,E1 -22453.291,E2 -22453.291} C_VEL
LIN {X 0,Y 223.566,Z 584.384,A -85,B 0,C 180,E1 -22456.306,E2 -22456.306} C_VEL
LIN {X 0,Y 223.481,Z 583.995,A -85,B 0,C 180,E1 -22459.004,E2 -22459.004} C_VEL
LIN {X 0,Y 222.633,Z 584.766,A -85,B 0,C 180,E1 -22462.111,E2 -22462.111} C_VEL
LIN {X 0,Y 221.743,Z 585.46,A -85,B 0,C 180,E1 -22462.973,E2 -22462.973} C_VEL
LIN {X 0,Y 212.76,Z 590.707,A -85,B 0,C 180,E1 -22465.837,E2 -22465.837} C_VEL
LIN {X 0,Y 204.582,Z 594.654,A -85,B 0,C 180,E1 -22468.983,E2 -22468.983} C_VEL
LIN {X 0,Y 197.372,Z 597.246,A -85,B 0,C 180,E1 -22472.426,E2 -22472.426} C_VEL
LIN {X 0,Y 191.122,Z 598.603,A -85,B 0,C 180,E1 -22476.141,E2 -22476.141} C_VEL
LIN {X 0,Y 186.003,Z 598.753,A -85,B 0,C 180,E1 -22480.12,E2 -22480.12} C_VEL
LIN {X 0,Y 182.057,Z 597.652,A -85,B 0,C 180,E1 -22484.323,E2 -22484.323} C_VEL
LIN {X 0,Y 179.069,Z 595.268,A -85,B 0,C 180,E1 -22488.683,E2 -22488.683} C_VEL
LIN {X 0,Y 177.499,Z 591.55,A -85,B 0,C 180,E1 -22493.179,E2 -22493.179} C_VEL
LIN {X 0,Y 176.836,Z 587.835,A -85,B 0,C 180,E1 -22496.583,E2 -22496.583} C_VEL
LIN {X 0,Y 176.529,Z 583.221,A -85,B 0,C 180,E1 -22500.001,E2 -22500.001} C_VEL
LIN {X 0,Y 176.638,Z 576.421,A -85,B 0,C 180,E1 -22503.993,E2 -22503.993} C_VEL
LIN {X 0,Y 177.169,Z 567.998,A -85,B 0,C 180,E1 -22507.981,E2 -22507.981} C_VEL
LIN {X 0,Y 177.893,Z 559.074,A -85,B 0,C 180,E1 -22511.393,E2 -22511.393} C_VEL
LIN {X 0,Y 178.84,Z 550.109,A -85,B 0,C 180,E1 -22514.219,E2 -22514.219} C_VEL
LIN {X 0,Y 180.174,Z 539.496,A -85,B 0,C 180,E1 -22517.011,E2 -22517.011} C_VEL
LIN {X 0,Y 181.579,Z 527.947,A -85,B 0,C 180,E1 -22519.502,E2 -22519.502} C_VEL
LIN {X 0,Y 182.054,Z 523.525,A -85,B 0,C 180,E1 -22520.331,E2 -22520.331} C_VEL
LIN {X 0,Y 180.377,Z 513.243,A -85,B 0,C 180,E1 -22522.036,E2 -22522.036} C_VEL
LIN {X 0,Y 177.997,Z 498.653,A -85,B 0,C 180,E1 -22524.017,E2 -22524.017} C_VEL
LIN {X 0,Y 177.3,Z 494.399,A -85,B 0,C 180,E1 -22524.511,E2 -22524.511} C_VEL
LIN {X 0,Y 177.646,Z 494.355,A -85,B 0,C 180,E1 -22529.498,E2 -22529.498} C_VEL
LIN {X 0,Y 178.096,Z 494.296,A -85,B 0,C 180,E1 -22534.033,E2 -22534.033} C_VEL
LIN {X 0,Y 178.348,Z 494.267,A -85,B 0,C 180,E1 -22539.088,E2 -22539.088} C_VEL
LIN {X 0,Y 178.397,Z 494.258,A -85,B 0,C 180,E1 -22542.047,E2 -22542.047} C_VEL
LIN {X 0,Y 178.405,Z 494.261,A -85,B 0,C 180,E1 -22545.162,E2 -22545.162} C_VEL
LIN {X 0,Y 178.415,Z 494.259,A -85,B 0,C 180,E1 -22548.456,E2 -22548.456} C_VEL
LIN {X 0,Y 178.468,Z 494.251,A -85,B 0,C 180,E1 -22551.962,E2 -22551.962} C_VEL
LIN {X 0,Y 178.495,Z 494.249,A -85,B 0,C 180,E1 -22556.548,E2 -22556.548} C_VEL
LIN {X 0,Y 178.527,Z 494.242,A -85,B 0,C 180,E1 -22560.006,E2 -22560.006} C_VEL
LIN {X 0,Y 178.539,Z 494.244,A -85,B 0,C 180,E1 -22564.875,E2 -22564.875} C_VEL
LIN {X 0,Y 178.628,Z 494.233,A -85,B 0,C 180,E1 -22570.783,E2 -22570.783} C_VEL
LIN {X 0,Y 178.664,Z 494.225,A -85,B 0,C 180,E1 -22576.348,E2 -22576.348} C_VEL
LIN {X 0,Y 178.916,Z 494.197,A -85,B 0,C 180,E1 -22580.959,E2 -22580.959} C_VEL
LIN {X 0,Y 179.157,Z 494.166,A -85,B 0,C 180,E1 -22587.751,E2 -22587.751} C_VEL
LIN {X 0,Y 179.374,Z 494.143,A -85,B 0,C 180,E1 -22590,E2 -22590} C_VEL
LIN {X 0,Y 178.866,Z 494.2,A -85,B 0,C 180,E1 -22594.507,E2 -22594.507} C_VEL
LIN {X 0,Y 178.912,Z 494.198,A -85,B 0,C 180,E1 -22599.04,E2 -22599.04} C_VEL
LIN {X 0,Y 178.663,Z 494.225,A -85,B 0,C 180,E1 -22603.651,E2 -22603.651} C_VEL
LIN {X 0,Y 178.627,Z 494.233,A -85,B 0,C 180,E1 -22609.216,E2 -22609.216} C_VEL
LIN {X 0,Y 178.537,Z 494.244,A -85,B 0,C 180,E1 -22615.124,E2 -22615.124} C_VEL
LIN {X 0,Y 178.482,Z 494.246,A -85,B 0,C 180,E1 -22620.79,E2 -22620.79} C_VEL
LIN {X 0,Y 178.499,Z 494.25,A -85,B 0,C 180,E1 -22624.224,E2 -22624.224} C_VEL
LIN {X 0,Y 178.42,Z 494.255,A -85,B 0,C 180,E1 -22629.067,E2 -22629.067} C_VEL
LIN {X 0,Y 178.405,Z 494.262,A -85,B 0,C 180,E1 -22632.043,E2 -22632.043} C_VEL
LIN {X 0,Y 178.4,Z 494.262,A -85,B 0,C 180,E1 -22635.161,E2 -22635.161} C_VEL
LIN {X 0,Y 178.405,Z 494.256,A -85,B 0,C 180,E1 -22638.458,E2 -22638.458} C_VEL
LIN {X 0,Y 178.424,Z 494.26,A -85,B 0,C 180,E1 -22643.782,E2 -22643.782} C_VEL
LIN {X 0,Y 178.489,Z 494.246,A -85,B 0,C 180,E1 -22646.546,E2 -22646.546} C_VEL
LIN {X 0,Y 178.524,Z 494.247,A -85,B 0,C 180,E1 -22650.005,E2 -22650.005} C_VEL
LIN {X 0,Y 178.535,Z 494.242,A -85,B 0,C 180,E1 -22654.875,E2 -22654.875} C_VEL
LIN {X 0,Y 178.624,Z 494.233,A -85,B 0,C 180,E1 -22660.783,E2 -22660.783} C_VEL
LIN {X 0,Y 178.682,Z 494.225,A -85,B 0,C 180,E1 -22666.349,E2 -22666.349} C_VEL
LIN {X 0,Y 178.979,Z 494.189,A -85,B 0,C 180,E1 -22670.963,E2 -22670.963} C_VEL
LIN {X 0,Y 179.155,Z 494.169,A -85,B 0,C 180,E1 -22677.751,E2 -22677.751} C_VEL
LIN {X 0,Y 179.371,Z 494.139,A -85,B 0,C 180,E1 -22679.999,E2 -22679.999} C_VEL
LIN {X 0,Y 178.876,Z 494.201,A -85,B 0,C 180,E1 -22684.506,E2 -22684.506} C_VEL
LIN {X 0,Y 178.979,Z 494.189,A -85,B 0,C 180,E1 -22689.036,E2 -22689.036} C_VEL
LIN {X 0,Y 178.688,Z 494.227,A -85,B 0,C 180,E1 -22693.649,E2 -22693.649} C_VEL
LIN {X 0,Y 178.671,Z 494.225,A -85,B 0,C 180,E1 -22698.341,E2 -22698.341} C_VEL
LIN {X 0,Y 178.513,Z 494.249,A -85,B 0,C 180,E1 -22703.184,E2 -22703.184} C_VEL
LIN {X 0,Y 178.485,Z 494.246,A -85,B 0,C 180,E1 -22708.197,E2 -22708.197} C_VEL
LIN {X 0,Y 178.476,Z 494.251,A -85,B 0,C 180,E1 -22710.791,E2 -22710.791} C_VEL
LIN {X 0,Y 178.483,Z 494.25,A -85,B 0,C 180,E1 -22714.219,E2 -22714.219} C_VEL
LIN {X 0,Y 178.514,Z 494.246,A -85,B 0,C 180,E1 -22719.043,E2 -22719.043} C_VEL
LIN {X 0,Y 178.666,Z 494.228,A -85,B 0,C 180,E1 -22721.967,E2 -22721.967} C_VEL
LIN {X 0,Y 178.925,Z 494.306,A -85,B 0,C 180,E1 -22725.192,E2 -22725.192} C_VEL
LIN {X 0,Y 179.677,Z 498.109,A -85,B 0,C 180,E1 -22729.806,E2 -22729.806} C_VEL
LIN {X 0,Y 180.047,Z 500.636,A -85,B 0,C 180,E1 -22732.794,E2 -22732.794} C_VEL
LIN {X 0,Y 179.583,Z 502.783,A -85,B 0,C 180,E1 -22735.269,E2 -22735.269} C_VEL
LIN {X 0,Y 178.39,Z 506.945,A -85,B 0,C 180,E1 -22740.081,E2 -22740.081} C_VEL
LIN {X 0,Y 177.468,Z 511.072,A -85,B 0,C 180,E1 -22744.838,E2 -22744.838} C_VEL
LIN {X 0,Y 177.722,Z 524.431,A -85,B 0,C 180,E1 -22746.328,E2 -22746.328} C_VEL
LIN {X 0,Y 178.536,Z 536.418,A -85,B 0,C 180,E1 -22748.04,E2 -22748.04} C_VEL
LIN {X 0,Y 179.764,Z 549.878,A -85,B 0,C 180,E1 -22750.433,E2 -22750.433} C_VEL
LIN {X 0,Y 180.73,Z 558.081,A -85,B 0,C 180,E1 -22752.168,E2 -22752.168} C_VEL
LIN {X 0,Y 179.565,Z 567.781,A -85,B 0,C 180,E1 -22754.682,E2 -22754.682} C_VEL
LIN {X 0,Y 178.723,Z 576.865,A -85,B 0,C 180,E1 -22757.51,E2 -22757.51} C_VEL
LIN {X 0,Y 178.089,Z 585.788,A -85,B 0,C 180,E1 -22760.918,E2 -22760.918} C_VEL
LIN {X 0,Y 177.865,Z 593.068,A -85,B 0,C 180,E1 -22764.331,E2 -22764.331} C_VEL
LIN {X 0,Y 177.826,Z 598.816,A -85,B 0,C 180,E1 -22767.735,E2 -22767.735} C_VEL
LIN {X 0,Y 177.846,Z 601.95,A -85,B 0,C 180,E1 -22770,E2 -22770} C_VEL
LIN {X 0,Y 177.227,Z 605.533,A -85,B 0,C 180,E1 -22773.411,E2 -22773.411} C_VEL
LIN {X 0,Y 176.905,Z 608.169,A -85,B 0,C 180,E1 -22776.845,E2 -22776.845} C_VEL
LIN {X 0,Y 177.318,Z 610.495,A -85,B 0,C 180,E1 -22781.431,E2 -22781.431} C_VEL
LIN {X 0,Y 178.854,Z 611.561,A -85,B 0,C 180,E1 -22785.966,E2 -22785.966} C_VEL
LIN {X 0,Y 181.962,Z 611.491,A -85,B 0,C 180,E1 -22790.342,E2 -22790.342} C_VEL
LIN {X 0,Y 186.245,Z 610.238,A -85,B 0,C 180,E1 -22794.525,E2 -22794.525} C_VEL
LIN {X 0,Y 191.7,Z 607.85,A -85,B 0,C 180,E1 -22798.464,E2 -22798.464} C_VEL
LIN {X 0,Y 193.833,Z 606.779,A -85,B 0,C 180,E1 -22799.679,E2 -22799.679} C_VEL
LIN {X 0,Y 196.067,Z 605.446,A -85,B 0,C 180,E1 -22801.24,E2 -22801.24} C_VEL
LIN {X 0,Y 200.907,Z 601.048,A -85,B 0,C 180,E1 -22806.027,E2 -22806.027} C_VEL
LIN {X 0,Y 203.483,Z 599.188,A -85,B 0,C 180,E1 -22807.428,E2 -22807.428} C_VEL
LIN {X 0,Y 204.583,Z 598.5,A -85,B 0,C 180,E1 -22807.842,E2 -22807.842} C_VEL
LIN {X 0,Y 207.446,Z 596.74,A -85,B 0,C 180,E1 -22808.812,E2 -22808.812} C_VEL
LIN {X 0,Y 209.426,Z 595.339,A -85,B 0,C 180,E1 -22809.614,E2 -22809.614} C_VEL
LIN {X 0,Y 213.966,Z 591.601,A -85,B 0,C 180,E1 -22812.327,E2 -22812.327} C_VEL
LIN {X 0,Y 215.314,Z 590.417,A -85,B 0,C 180,E1 -22813.272,E2 -22813.272} C_VEL
LIN {X 0,Y 216.479,Z 589.284,A -85,B 0,C 180,E1 -22814.42,E2 -22814.42} C_VEL
LIN {X 0,Y 216.947,Z 588.627,A -85,B 0,C 180,E1 -22815.455,E2 -22815.455} C_VEL
LIN {X 0,Y 217.447,Z 587.882,A -85,B 0,C 180,E1 -22817.256,E2 -22817.256} C_VEL
LIN {X 0,Y 217.161,Z 587.754,A -85,B 0,C 180,E1 -22819.665,E2 -22819.665} C_VEL
LIN {X 0,Y 216.353,Z 588.256,A -85,B 0,C 180,E1 -22821.889,E2 -22821.889} C_VEL
LIN {X 0,Y 207.157,Z 592.945,A -85,B 0,C 180,E1 -22824.779,E2 -22824.779} C_VEL
LIN {X 0,Y 198.693,Z 596.365,A -85,B 0,C 180,E1 -22827.957,E2 -22827.957} C_VEL
LIN {X 0,Y 191.227,Z 598.521,A -85,B 0,C 180,E1 -22831.46,E2 -22831.46} C_VEL
LIN {X 0,Y 184.721,Z 599.478,A -85,B 0,C 180,E1 -22835.26,E2 -22835.26} C_VEL
LIN {X 0,Y 179.368,Z 599.209,A -85,B 0,C 180,E1 -22839.352,E2 -22839.352} C_VEL
LIN {X 0,Y 175.231,Z 597.718,A -85,B 0,C 180,E1 -22843.695,E2 -22843.695} C_VEL
LIN {X 0,Y 172.143,Z 594.983,A -85,B 0,C 180,E1 -22848.222,E2 -22848.222} C_VEL
LIN {X 0,Y 170.493,Z 590.975,A -85,B 0,C 180,E1 -22852.897,E2 -22852.897} C_VEL
LIN {X 0,Y 169.817,Z 586.963,A -85,B 0,C 180,E1 -22856.441,E2 -22856.441} C_VEL
LIN {X 0,Y 169.527,Z 582.037,A -85,B 0,C 180,E1 -22860.001,E2 -22860.001} C_VEL
LIN {X 0,Y 169.62,Z 576.088,A -85,B 0,C 180,E1 -22863.564,E2 -22863.564} C_VEL
LIN {X 0,Y 170.113,Z 567.607,A -85,B 0,C 180,E1 -22867.657,E2 -22867.657} C_VEL
LIN {X 0,Y 170.843,Z 558.37,A -85,B 0,C 180,E1 -22871.269,E2 -22871.269} C_VEL
LIN {X 0,Y 171.802,Z 549.367,A -85,B 0,C 180,E1 -22874.209,E2 -22874.209} C_VEL
LIN {X 0,Y 173.124,Z 538.619,A -85,B 0,C 180,E1 -22877.117,E2 -22877.117} C_VEL
LIN {X 0,Y 174.585,Z 526.776,A -85,B 0,C 180,E1 -22879.703,E2 -22879.703} C_VEL
LIN {X 0,Y 174.798,Z 522.035,A -85,B 0,C 180,E1 -22880.598,E2 -22880.598} C_VEL
LIN {X 0,Y 172.476,Z 509.067,A -85,B 0,C 180,E1 -22882.738,E2 -22882.738} C_VEL
LIN {X 0,Y 170.26,Z 495.276,A -85,B 0,C 180,E1 -22884.569,E2 -22884.569} C_VEL
LIN {X 0,Y 170.662,Z 495.227,A -85,B 0,C 180,E1 -22890.139,E2 -22890.139} C_VEL
LIN {X 0,Y 171.08,Z 495.172,A -85,B 0,C 180,E1 -22895.109,E2 -22895.109} C_VEL
LIN {X 0,Y 171.29,Z 495.147,A -85,B 0,C 180,E1 -22898.778,E2 -22898.778} C_VEL
LIN {X 0,Y 171.336,Z 495.139,A -85,B 0,C 180,E1 -22902.409,E2 -22902.409} C_VEL
LIN {X 0,Y 171.344,Z 495.14,A -85,B 0,C 180,E1 -22907.588,E2 -22907.588} C_VEL
LIN {X 0,Y 171.417,Z 495.129,A -85,B 0,C 180,E1 -22912.048,E2 -22912.048} C_VEL
LIN {X 0,Y 171.415,Z 495.132,A -85,B 0,C 180,E1 -22915.086,E2 -22915.086} C_VEL
LIN {X 0,Y 171.454,Z 495.126,A -85,B 0,C 180,E1 -22920.535,E2 -22920.535} C_VEL
LIN {X 0,Y 171.462,Z 495.126,A -85,B 0,C 180,E1 -22925.802,E2 -22925.802} C_VEL
LIN {X 0,Y 171.584,Z 495.11,A -85,B 0,C 180,E1 -22930.872,E2 -22930.872} C_VEL
LIN {X 0,Y 171.582,Z 495.11,A -85,B 0,C 180,E1 -22935.773,E2 -22935.773} C_VEL
LIN {X 0,Y 171.852,Z 495.078,A -85,B 0,C 180,E1 -22940.585,E2 -22940.585} C_VEL
LIN {X 0,Y 171.82,Z 495.077,A -85,B 0,C 180,E1 -22945.307,E2 -22945.307} C_VEL
LIN {X 0,Y 172.337,Z 495.02,A -85,B 0,C 180,E1 -22949.999,E2 -22949.999} C_VEL
LIN {X 0,Y 171.814,Z 495.078,A -85,B 0,C 180,E1 -22954.692,E2 -22954.692} C_VEL
LIN {X 0,Y 171.85,Z 495.078,A -85,B 0,C 180,E1 -22959.415,E2 -22959.415} C_VEL
LIN {X 0,Y 171.581,Z 495.11,A -85,B 0,C 180,E1 -22964.226,E2 -22964.226} C_VEL
LIN {X 0,Y 171.548,Z 495.116,A -85,B 0,C 180,E1 -22969.562,E2 -22969.562} C_VEL
LIN {X 0,Y 171.472,Z 495.126,A -85,B 0,C 180,E1 -22975.616,E2 -22975.616} C_VEL
LIN {X 0,Y 171.444,Z 495.122,A -85,B 0,C 180,E1 -22980.586,E2 -22980.586} C_VEL
LIN {X 0,Y 171.409,Z 495.132,A -85,B 0,C 180,E1 -22985.03,E2 -22985.03} C_VEL
LIN {X 0,Y 171.382,Z 495.131,A -85,B 0,C 180,E1 -22988.816,E2 -22988.816} C_VEL
LIN {X 0,Y 171.329,Z 495.143,A -85,B 0,C 180,E1 -22994.214,E2 -22994.214} C_VEL
LIN {X 0,Y 171.337,Z 495.137,A -85,B 0,C 180,E1 -22998.981,E2 -22998.981} C_VEL
LIN {X 0,Y 171.388,Z 495.136,A -85,B 0,C 180,E1 -23002.04,E2 -23002.04} C_VEL
LIN {X 0,Y 171.399,Z 495.133,A -85,B 0,C 180,E1 -23005.091,E2 -23005.091} C_VEL
LIN {X 0,Y 171.45,Z 495.127,A -85,B 0,C 180,E1 -23010.534,E2 -23010.534} C_VEL
LIN {X 0,Y 171.459,Z 495.123,A -85,B 0,C 180,E1 -23015.801,E2 -23015.801} C_VEL
LIN {X 0,Y 171.58,Z 495.111,A -85,B 0,C 180,E1 -23020.871,E2 -23020.871} C_VEL
LIN {X 0,Y 171.595,Z 495.108,A -85,B 0,C 180,E1 -23025.774,E2 -23025.774} C_VEL
LIN {X 0,Y 171.911,Z 495.069,A -85,B 0,C 180,E1 -23030.588,E2 -23030.588} C_VEL
LIN {X 0,Y 171.827,Z 495.079,A -85,B 0,C 180,E1 -23035.307,E2 -23035.307} C_VEL
LIN {X 0,Y 172.334,Z 495.016,A -85,B 0,C 180,E1 -23039.999,E2 -23039.999} C_VEL
LIN {X 0,Y 171.826,Z 495.079,A -85,B 0,C 180,E1 -23044.692,E2 -23044.692} C_VEL
LIN {X 0,Y 171.91,Z 495.069,A -85,B 0,C 180,E1 -23049.411,E2 -23049.411} C_VEL
LIN {X 0,Y 171.613,Z 495.107,A -85,B 0,C 180,E1 -23054.224,E2 -23054.224} C_VEL
LIN {X 0,Y 171.557,Z 495.11,A -85,B 0,C 180,E1 -23059.574,E2 -23059.574} C_VEL
LIN {X 0,Y 171.468,Z 495.125,A -85,B 0,C 180,E1 -23065.616,E2 -23065.616} C_VEL
LIN {X 0,Y 171.439,Z 495.127,A -85,B 0,C 180,E1 -23070.585,E2 -23070.585} C_VEL
LIN {X 0,Y 171.407,Z 495.134,A -85,B 0,C 180,E1 -23075.031,E2 -23075.031} C_VEL
LIN {X 0,Y 171.482,Z 495.121,A -85,B 0,C 180,E1 -23078.859,E2 -23078.859} C_VEL
LIN {X 0,Y 171.87,Z 495.082,A -85,B 0,C 180,E1 -23085.022,E2 -23085.022} C_VEL
LIN {X 0,Y 171.963,Z 495.402,A -85,B 0,C 180,E1 -23085.991,E2 -23085.991} C_VEL
LIN {X 0,Y 172.708,Z 499.096,A -85,B 0,C 180,E1 -23090.638,E2 -23090.638} C_VEL
LIN {X 0,Y 172.916,Z 500.547,A -85,B 0,C 180,E1 -23092.436,E2 -23092.436} C_VEL
LIN {X 0,Y 172.467,Z 502.859,A -85,B 0,C 180,E1 -23095.216,E2 -23095.216} C_VEL
LIN {X 0,Y 171.155,Z 507.193,A -85,B 0,C 180,E1 -23100.479,E2 -23100.479} C_VEL
LIN {X 0,Y 170.4,Z 510.703,A -85,B 0,C 180,E1 -23104.736,E2 -23104.736} C_VEL
LIN {X 0,Y 170.615,Z 524.227,A -85,B 0,C 180,E1 -23106.321,E2 -23106.321} C_VEL
LIN {X 0,Y 171.535,Z 537.63,A -85,B 0,C 180,E1 -23108.362,E2 -23108.362} C_VEL
LIN {X 0,Y 172.796,Z 550.56,A -85,B 0,C 180,E1 -23110.807,E2 -23110.807} C_VEL
LIN {X 0,Y 173.633,Z 557.4,A -85,B 0,C 180,E1 -23112.328,E2 -23112.328} C_VEL
LIN {X 0,Y 172.424,Z 568.137,A -85,B 0,C 180,E1 -23115.242,E2 -23115.242} C_VEL
LIN {X 0,Y 171.523,Z 578.622,A -85,B 0,C 180,E1 -23118.778,E2 -23118.778} C_VEL
LIN {X 0,Y 171.078,Z 586.599,A -85,B 0,C 180,E1 -23122.111,E2 -23122.111} C_VEL
LIN {X 0,Y 170.947,Z 593.865,A -85,B 0,C 180,E1 -23125.875,E2 -23125.875} C_VEL
LIN {X 0,Y 170.944,Z 598.453,A -85,B 0,C 180,E1 -23128.823,E2 -23128.823} C_VEL
LIN {X 0,Y 170.822,Z 601.481,A -85,B 0,C 180,E1 -23131.179,E2 -23131.179} C_VEL
LIN {X 0,Y 170.153,Z 604.897,A -85,B 0,C 180,E1 -23134.739,E2 -23134.739} C_VEL
LIN {X 0,Y 170.049,Z 608.204,A -85,B 0,C 180,E1 -23139.516,E2 -23139.516} C_VEL
LIN {X 0,Y 171.103,Z 610.159,A -85,B 0,C 180,E1 -23144.268,E2 -23144.268} C_VEL
LIN {X 0,Y 173.543,Z 610.965,A -85,B 0,C 180,E1 -23148.904,E2 -23148.904} C_VEL
LIN {X 0,Y 177.407,Z 610.641,A -85,B 0,C 180,E1 -23153.338,E2 -23153.338} C_VEL
LIN {X 0,Y 183.807,Z 608.722,A -85,B 0,C 180,E1 -23158.427,E2 -23158.427} C_VEL
LIN {X 0,Y 188.915,Z 606.645,A -85,B 0,C 180,E1 -23161.388,E2 -23161.388} C_VEL
LIN {X 0,Y 196.584,Z 602.957,A -85,B 0,C 180,E1 -23164.891,E2 -23164.891} C_VEL
LIN {X 0,Y 204.583,Z 598.5,A -85,B 0,C 180,E1 -23167.842,E2 -23167.842} C_VEL
LIN {X 0,Y 206.247,Z 597.282,A -85,B 0,C 180,E1 -23168.758,E2 -23168.758} C_VEL
LIN {X 0,Y 206.936,Z 596.374,A -85,B 0,C 180,E1 -23169.814,E2 -23169.814} C_VEL
LIN {X 0,Y 207.747,Z 594.403,A -85,B 0,C 180,E1 -23172.796,E2 -23172.796} C_VEL
LIN {X 0,Y 208.554,Z 593.729,A -85,B 0,C 180,E1 -23173.495,E2 -23173.495} C_VEL
LIN {X 0,Y 210.021,Z 592.594,A -85,B 0,C 180,E1 -23174.647,E2 -23174.647} C_VEL
LIN {X 0,Y 210.604,Z 591.99,A -85,B 0,C 180,E1 -23175.51,E2 -23175.51} C_VEL
LIN {X 0,Y 211.099,Z 591.327,A -85,B 0,C 180,E1 -23177.092,E2 -23177.092} C_VEL
LIN {X 0,Y 211.131,Z 591.096,A -85,B 0,C 180,E1 -23178.261,E2 -23178.261} C_VEL
LIN {X 0,Y 210.548,Z 591.186,A -85,B 0,C 180,E1 -23180.639,E2 -23180.639} C_VEL
LIN {X 0,Y 206.322,Z 593.101,A -85,B 0,C 180,E1 -23182.184,E2 -23182.184} C_VEL
LIN {X 0,Y 197.121,Z 596.658,A -85,B 0,C 180,E1 -23185.219,E2 -23185.219} C_VEL
LIN {X 0,Y 188.841,Z 598.96,A -85,B 0,C 180,E1 -23188.599,E2 -23188.599} C_VEL
LIN {X 0,Y 181.582,Z 600.083,A -85,B 0,C 180,E1 -23192.326,E2 -23192.326} C_VEL
LIN {X 0,Y 175.45,Z 600.034,A -85,B 0,C 180,E1 -23196.387,E2 -23196.387} C_VEL
LIN {X 0,Y 170.473,Z 598.778,A -85,B 0,C 180,E1 -23200.743,E2 -23200.743} C_VEL
LIN {X 0,Y 166.645,Z 596.286,A -85,B 0,C 180,E1 -23205.343,E2 -23205.343} C_VEL
LIN {X 0,Y 164.159,Z 592.547,A -85,B 0,C 180,E1 -23210.14,E2 -23210.14} C_VEL
LIN {X 0,Y 162.998,Z 587.476,A -85,B 0,C 180,E1 -23215.054,E2 -23215.054} C_VEL
LIN {X 0,Y 162.562,Z 582.594,A -85,B 0,C 180,E1 -23218.762,E2 -23218.762} C_VEL
LIN {X 0,Y 162.612,Z 575.602,A -85,B 0,C 180,E1 -23223.097,E2 -23223.097} C_VEL
LIN {X 0,Y 163.083,Z 566.885,A -85,B 0,C 180,E1 -23227.429,E2 -23227.429} C_VEL
LIN {X 0,Y 163.803,Z 557.632,A -85,B 0,C 180,E1 -23231.133,E2 -23231.133} C_VEL
LIN {X 0,Y 164.891,Z 547.396,A -85,B 0,C 180,E1 -23234.502,E2 -23234.502} C_VEL
LIN {X 0,Y 166.228,Z 536.204,A -85,B 0,C 180,E1 -23237.533,E2 -23237.533} C_VEL
LIN {X 0,Y 167.59,Z 525.605,A -85,B 0,C 180,E1 -23239.906,E2 -23239.906} C_VEL
LIN {X 0,Y 167.7,Z 522.557,A -85,B 0,C 180,E1 -23240.499,E2 -23240.499} C_VEL
LIN {X 0,Y 165.486,Z 510.176,A -85,B 0,C 180,E1 -23242.636,E2 -23242.636} C_VEL
LIN {X 0,Y 163.218,Z 496.153,A -85,B 0,C 180,E1 -23244.57,E2 -23244.57} C_VEL
LIN {X 0,Y 163.687,Z 496.092,A -85,B 0,C 180,E1 -23251.014,E2 -23251.014} C_VEL
LIN {X 0,Y 164.036,Z 496.05,A -85,B 0,C 180,E1 -23255.506,E2 -23255.506} C_VEL
LIN {X 0,Y 164.231,Z 496.027,A -85,B 0,C 180,E1 -23259.935,E2 -23259.935} C_VEL
LIN {X 0,Y 164.283,Z 496.017,A -85,B 0,C 180,E1 -23263.342,E2 -23263.342} C_VEL
LIN {X 0,Y 164.296,Z 496.019,A -85,B 0,C 180,E1 -23266.809,E2 -23266.809} C_VEL
LIN {X 0,Y 164.309,Z 496.013,A -85,B 0,C 180,E1 -23270.348,E2 -23270.348} C_VEL
LIN {X 0,Y 164.347,Z 496.014,A -85,B 0,C 180,E1 -23274.342,E2 -23274.342} C_VEL
LIN {X 0,Y 164.395,Z 496,A -85,B 0,C 180,E1 -23279.135,E2 -23279.135} C_VEL
LIN {X 0,Y 164.421,Z 496.003,A -85,B 0,C 180,E1 -23284.694,E2 -23284.694} C_VEL
LIN {X 0,Y 164.489,Z 495.993,A -85,B 0,C 180,E1 -23290.051,E2 -23290.051} C_VEL
LIN {X 0,Y 164.529,Z 495.987,A -85,B 0,C 180,E1 -23295.149,E2 -23295.149} C_VEL
LIN {X 0,Y 164.773,Z 495.961,A -85,B 0,C 180,E1 -23300.176,E2 -23300.176} C_VEL
LIN {X 0,Y 164.836,Z 495.951,A -85,B 0,C 180,E1 -23302.651,E2 -23302.651} C_VEL
LIN {X 0,Y 165.052,Z 495.922,A -85,B 0,C 180,E1 -23307.559,E2 -23307.559} C_VEL
LIN {X 0,Y 165.299,Z 495.896,A -85,B 0,C 180,E1 -23309.999,E2 -23309.999} C_VEL
LIN {X 0,Y 164.763,Z 495.956,A -85,B 0,C 180,E1 -23314.893,E2 -23314.893} C_VEL
LIN {X 0,Y 164.831,Z 495.951,A -85,B 0,C 180,E1 -23317.348,E2 -23317.348} C_VEL
LIN {X 0,Y 164.706,Z 495.966,A -85,B 0,C 180,E1 -23321.06,E2 -23321.06} C_VEL
LIN {X 0,Y 164.488,Z 495.995,A -85,B 0,C 180,E1 -23327.402,E2 -23327.402} C_VEL
LIN {X 0,Y 164.477,Z 495.995,A -85,B 0,C 180,E1 -23329.988,E2 -23329.988} C_VEL
LIN {X 0,Y 164.397,Z 496.007,A -85,B 0,C 180,E1 -23336.133,E2 -23336.133} C_VEL
LIN {X 0,Y 164.379,Z 496.003,A -85,B 0,C 180,E1 -23341.228,E2 -23341.228} C_VEL
LIN {X 0,Y 164.315,Z 496.015,A -85,B 0,C 180,E1 -23346.783,E2 -23346.783} C_VEL
LIN {X 0,Y 164.301,Z 496.014,A -85,B 0,C 180,E1 -23349.913,E2 -23349.913} C_VEL
LIN {X 0,Y 164.281,Z 496.021,A -85,B 0,C 180,E1 -23353.341,E2 -23353.341} C_VEL
LIN {X 0,Y 164.293,Z 496.016,A -85,B 0,C 180,E1 -23356.808,E2 -23356.808} C_VEL
LIN {X 0,Y 164.296,Z 496.017,A -85,B 0,C 180,E1 -23360.351,E2 -23360.351} C_VEL
LIN {X 0,Y 164.331,Z 496.013,A -85,B 0,C 180,E1 -23364.348,E2 -23364.348} C_VEL
LIN {X 0,Y 164.392,Z 496.004,A -85,B 0,C 180,E1 -23369.134,E2 -23369.134} C_VEL
LIN {X 0,Y 164.417,Z 496,A -85,B 0,C 180,E1 -23374.693,E2 -23374.693} C_VEL
LIN {X 0,Y 164.485,Z 495.996,A -85,B 0,C 180,E1 -23380.05,E2 -23380.05} C_VEL
LIN {X 0,Y 164.537,Z 495.983,A -85,B 0,C 180,E1 -23385.15,E2 -23385.15} C_VEL
LIN {X 0,Y 164.853,Z 495.949,A -85,B 0,C 180,E1 -23390.181,E2 -23390.181} C_VEL
LIN {X 0,Y 164.863,Z 495.944,A -85,B 0,C 180,E1 -23392.652,E2 -23392.652} C_VEL
LIN {X 0,Y 165.052,Z 495.927,A -85,B 0,C 180,E1 -23397.559,E2 -23397.559} C_VEL
LIN {X 0,Y 165.296,Z 495.892,A -85,B 0,C 180,E1 -23399.999,E2 -23399.999} C_VEL
LIN {X 0,Y 164.776,Z 495.958,A -85,B 0,C 180,E1 -23404.893,E2 -23404.893} C_VEL
LIN {X 0,Y 164.862,Z 495.95,A -85,B 0,C 180,E1 -23407.347,E2 -23407.347} C_VEL
LIN {X 0,Y 164.78,Z 495.954,A -85,B 0,C 180,E1 -23411.198,E2 -23411.198} C_VEL
LIN {X 0,Y 164.52,Z 495.991,A -85,B 0,C 180,E1 -23417.399,E2 -23417.399} C_VEL
LIN {X 0,Y 164.475,Z 495.992,A -85,B 0,C 180,E1 -23419.989,E2 -23419.989} C_VEL
LIN {X 0,Y 164.392,Z 496.005,A -85,B 0,C 180,E1 -23426.133,E2 -23426.133} C_VEL
LIN {X 0,Y 164.373,Z 496.009,A -85,B 0,C 180,E1 -23431.227,E2 -23431.227} C_VEL
LIN {X 0,Y 164.355,Z 496.008,A -85,B 0,C 180,E1 -23436.773,E2 -23436.773} C_VEL
LIN {X 0,Y 164.44,Z 496,A -85,B 0,C 180,E1 -23439.872,E2 -23439.872} C_VEL
LIN {X 0,Y 164.912,Z 495.99,A -85,B 0,C 180,E1 -23446.217,E2 -23446.217} C_VEL
LIN {X 0,Y 165.584,Z 499.212,A -85,B 0,C 180,E1 -23450.458,E2 -23450.458} C_VEL
LIN {X 0,Y 165.769,Z 500.456,A -85,B 0,C 180,E1 -23452.067,E2 -23452.067} C_VEL
LIN {X 0,Y 165.396,Z 502.83,A -85,B 0,C 180,E1 -23455.081,E2 -23455.081} C_VEL
LIN {X 0,Y 164.056,Z 507.06,A -85,B 0,C 180,E1 -23460.486,E2 -23460.486} C_VEL
LIN {X 0,Y 163.314,Z 510.208,A -85,B 0,C 180,E1 -23464.572,E2 -23464.572} C_VEL
LIN {X 0,Y 163.55,Z 524.728,A -85,B 0,C 180,E1 -23466.412,E2 -23466.412} C_VEL
LIN {X 0,Y 164.486,Z 537.988,A -85,B 0,C 180,E1 -23468.563,E2 -23468.563} C_VEL
LIN {X 0,Y 165.78,Z 550.857,A -85,B 0,C 180,E1 -23471.141,E2 -23471.141} C_VEL
LIN {X 0,Y 166.548,Z 556.72,A -85,B 0,C 180,E1 -23472.503,E2 -23472.503} C_VEL
LIN {X 0,Y 165.506,Z 566.428,A -85,B 0,C 180,E1 -23475.24,E2 -23475.24} C_VEL
LIN {X 0,Y 164.741,Z 575.728,A -85,B 0,C 180,E1 -23478.418,E2 -23478.418} C_VEL
LIN {X 0,Y 164.232,Z 584.289,A -85,B 0,C 180,E1 -23482.006,E2 -23482.006} C_VEL
LIN {X 0,Y 164.104,Z 591.488,A -85,B 0,C 180,E1 -23485.702,E2 -23485.702} C_VEL
LIN {X 0,Y 164.076,Z 596.353,A -85,B 0,C 180,E1 -23488.773,E2 -23488.773} C_VEL
LIN {X 0,Y 164.012,Z 599.504,A -85,B 0,C 180,E1 -23491.228,E2 -23491.228} C_VEL
LIN {X 0,Y 163.278,Z 603.174,A -85,B 0,C 180,E1 -23494.939,E2 -23494.939} C_VEL
LIN {X 0,Y 163.17,Z 606.729,A -85,B 0,C 180,E1 -23499.921,E2 -23499.921} C_VEL
LIN {X 0,Y 164.291,Z 609.01,A -85,B 0,C 180,E1 -23504.873,E2 -23504.873} C_VEL
LIN {X 0,Y 166.86,Z 610.127,A -85,B 0,C 180,E1 -23509.692,E2 -23509.692} C_VEL
LIN {X 0,Y 170.911,Z 610.161,A -85,B 0,C 180,E1 -23514.281,E2 -23514.281} C_VEL
LIN {X 0,Y 176.883,Z 608.919,A -85,B 0,C 180,E1 -23519.06,E2 -23519.06} C_VEL
LIN {X 0,Y 182.913,Z 606.975,A -85,B 0,C 180,E1 -23522.543,E2 -23522.543} C_VEL
LIN {X 0,Y 190.847,Z 603.758,A -85,B 0,C 180,E1 -23526.101,E2 -23526.101} C_VEL
LIN {X 0,Y 200.283,Z 599.132,A -85,B 0,C 180,E1 -23529.468,E2 -23529.468} C_VEL
LIN {X 0,Y 204.099,Z 596.939,A -85,B 0,C 180,E1 -23530.863,E2 -23530.863} C_VEL
LIN {X 0,Y 208.554,Z 593.729,A -85,B 0,C 180,E1 -23533.495,E2 -23533.495} C_VEL
LIN {X 0,Y 209.426,Z 592.944,A -85,B 0,C 180,E1 -23534.543,E2 -23534.543} C_VEL
LIN {X 0,Y 209.249,Z 592.679,A -85,B 0,C 180,E1 -23535.652,E2 -23535.652} C_VEL
LIN {X 0,Y 207.863,Z 592.929,A -85,B 0,C 180,E1 -23537.137,E2 -23537.137} C_VEL
LIN {X 0,Y 205.626,Z 593.655,A -85,B 0,C 180,E1 -23538.589,E2 -23538.589} C_VEL
LIN {X 0,Y 204.29,Z 594.118,A -85,B 0,C 180,E1 -23539.288,E2 -23539.288} C_VEL
LIN {X 0,Y 200.987,Z 595.346,A -85,B 0,C 180,E1 -23540.993,E2 -23540.993} C_VEL
LIN {X 0,Y 191.486,Z 598.366,A -85,B 0,C 180,E1 -23544.039,E2 -23544.039} C_VEL
LIN {X 0,Y 182.907,Z 600.207,A -85,B 0,C 180,E1 -23547.457,E2 -23547.457} C_VEL
LIN {X 0,Y 175.376,Z 600.887,A -85,B 0,C 180,E1 -23551.257,E2 -23551.257} C_VEL
LIN {X 0,Y 169.002,Z 600.407,A -85,B 0,C 180,E1 -23555.427,E2 -23555.427} C_VEL
LIN {X 0,Y 163.811,Z 598.766,A -85,B 0,C 180,E1 -23559.927,E2 -23559.927} C_VEL
LIN {X 0,Y 159.809,Z 595.938,A -85,B 0,C 180,E1 -23564.701,E2 -23564.701} C_VEL
LIN {X 0,Y 157.22,Z 591.848,A -85,B 0,C 180,E1 -23569.7,E2 -23569.7} C_VEL
LIN {X 0,Y 156.023,Z 586.378,A -85,B 0,C 180,E1 -23574.832,E2 -23574.832} C_VEL
LIN {X 0,Y 155.538,Z 579.333,A -85,B 0,C 180,E1 -23580.001,E2 -23580.001} C_VEL
LIN {X 0,Y 155.666,Z 572.684,A -85,B 0,C 180,E1 -23583.884,E2 -23583.884} C_VEL
LIN {X 0,Y 156.219,Z 563.633,A -85,B 0,C 180,E1 -23588.211,E2 -23588.211} C_VEL
LIN {X 0,Y 157.176,Z 553.279,A -85,B 0,C 180,E1 -23592.263,E2 -23592.263} C_VEL
LIN {X 0,Y 158.432,Z 542.058,A -85,B 0,C 180,E1 -23595.766,E2 -23595.766} C_VEL
LIN {X 0,Y 159.985,Z 529.695,A -85,B 0,C 180,E1 -23598.904,E2 -23598.904} C_VEL
LIN {X 0,Y 160.639,Z 523.867,A -85,B 0,C 180,E1 -23600.154,E2 -23600.154} C_VEL
LIN {X 0,Y 158.743,Z 512.693,A -85,B 0,C 180,E1 -23602.209,E2 -23602.209} C_VEL
LIN {X 0,Y 156.527,Z 499.437,A -85,B 0,C 180,E1 -23604.22,E2 -23604.22} C_VEL
LIN {X 0,Y 156.192,Z 497.028,A -85,B 0,C 180,E1 -23604.623,E2 -23604.623} C_VEL
LIN {X 0,Y 156.669,Z 496.966,A -85,B 0,C 180,E1 -23611.534,E2 -23611.534} C_VEL
LIN {X 0,Y 157.021,Z 496.926,A -85,B 0,C 180,E1 -23616.326,E2 -23616.326} C_VEL
LIN {X 0,Y 157.153,Z 496.905,A -85,B 0,C 180,E1 -23620.513,E2 -23620.513} C_VEL
LIN {X 0,Y 157.181,Z 496.905,A -85,B 0,C 180,E1 -23625.678,E2 -23625.678} C_VEL
LIN {X 0,Y 157.242,Z 496.893,A -85,B 0,C 180,E1 -23631.263,E2 -23631.263} C_VEL
LIN {X 0,Y 157.295,Z 496.892,A -85,B 0,C 180,E1 -23634.489,E2 -23634.489} C_VEL
LIN {X 0,Y 157.299,Z 496.887,A -85,B 0,C 180,E1 -23638.095,E2 -23638.095} C_VEL
LIN {X 0,Y 157.326,Z 496.887,A -85,B 0,C 180,E1 -23643.466,E2 -23643.466} C_VEL
LIN {X 0,Y 157.398,Z 496.875,A -85,B 0,C 180,E1 -23649.667,E2 -23649.667} C_VEL
LIN {X 0,Y 157.459,Z 496.869,A -85,B 0,C 180,E1 -23654.466,E2 -23654.466} C_VEL
LIN {X 0,Y 157.694,Z 496.841,A -85,B 0,C 180,E1 -23659.73,E2 -23659.73} C_VEL
LIN {X 0,Y 157.772,Z 496.831,A -85,B 0,C 180,E1 -23662.32,E2 -23662.32} C_VEL
LIN {X 0,Y 158.261,Z 496.773,A -85,B 0,C 180,E1 -23669.999,E2 -23669.999} C_VEL
LIN {X 0,Y 157.768,Z 496.832,A -85,B 0,C 180,E1 -23677.679,E2 -23677.679} C_VEL
LIN {X 0,Y 157.64,Z 496.846,A -85,B 0,C 180,E1 -23681.237,E2 -23681.237} C_VEL
LIN {X 0,Y 157.458,Z 496.869,A -85,B 0,C 180,E1 -23685.533,E2 -23685.533} C_VEL
LIN {X 0,Y 157.373,Z 496.877,A -85,B 0,C 180,E1 -23690.932,E2 -23690.932} C_VEL
LIN {X 0,Y 157.318,Z 496.888,A -85,B 0,C 180,E1 -23696.684,E2 -23696.684} C_VEL
LIN {X 0,Y 157.281,Z 496.891,A -85,B 0,C 180,E1 -23702.426,E2 -23702.426} C_VEL
LIN {X 0,Y 157.285,Z 496.891,A -85,B 0,C 180,E1 -23706.456,E2 -23706.456} C_VEL
LIN {X 0,Y 157.214,Z 496.901,A -85,B 0,C 180,E1 -23712.109,E2 -23712.109} C_VEL
LIN {X 0,Y 157.212,Z 496.897,A -85,B 0,C 180,E1 -23717.889,E2 -23717.889} C_VEL
LIN {X 0,Y 157.269,Z 496.896,A -85,B 0,C 180,E1 -23723.55,E2 -23723.55} C_VEL
LIN {X 0,Y 157.295,Z 496.889,A -85,B 0,C 180,E1 -23728.094,E2 -23728.094} C_VEL
LIN {X 0,Y 157.323,Z 496.888,A -85,B 0,C 180,E1 -23733.466,E2 -23733.466} C_VEL
LIN {X 0,Y 157.395,Z 496.88,A -85,B 0,C 180,E1 -23739.666,E2 -23739.666} C_VEL
LIN {X 0,Y 157.463,Z 496.863,A -85,B 0,C 180,E1 -23744.466,E2 -23744.466} C_VEL
LIN {X 0,Y 157.773,Z 496.832,A -85,B 0,C 180,E1 -23749.736,E2 -23749.736} C_VEL
LIN {X 0,Y 157.825,Z 496.82,A -85,B 0,C 180,E1 -23752.322,E2 -23752.322} C_VEL
LIN {X 0,Y 158.258,Z 496.769,A -85,B 0,C 180,E1 -23759.999,E2 -23759.999} C_VEL
LIN {X 0,Y 157.825,Z 496.825,A -85,B 0,C 180,E1 -23767.677,E2 -23767.677} C_VEL
LIN {X 0,Y 157.706,Z 496.835,A -85,B 0,C 180,E1 -23771.362,E2 -23771.362} C_VEL
LIN {X 0,Y 157.485,Z 496.869,A -85,B 0,C 180,E1 -23775.53,E2 -23775.53} C_VEL
LIN {X 0,Y 157.371,Z 496.877,A -85,B 0,C 180,E1 -23780.932,E2 -23780.932} C_VEL
LIN {X 0,Y 157.313,Z 496.887,A -85,B 0,C 180,E1 -23786.684,E2 -23786.684} C_VEL
LIN {X 0,Y 157.276,Z 496.893,A -85,B 0,C 180,E1 -23792.427,E2 -23792.427} C_VEL
LIN {X 0,Y 157.328,Z 496.883,A -85,B 0,C 180,E1 -23796.479,E2 -23796.479} C_VEL
LIN {X 0,Y 157.471,Z 496.869,A -85,B 0,C 180,E1 -23802.025,E2 -23802.025} C_VEL
LIN {X 0,Y 157.907,Z 496.896,A -85,B 0,C 180,E1 -23806.969,E2 -23806.969} C_VEL
LIN {X 0,Y 158.627,Z 500.327,A -85,B 0,C 180,E1 -23811.665,E2 -23811.665} C_VEL
LIN {X 0,Y 158.334,Z 502.639,A -85,B 0,C 180,E1 -23814.758,E2 -23814.758} C_VEL
LIN {X 0,Y 156.939,Z 506.895,A -85,B 0,C 180,E1 -23820.489,E2 -23820.489} C_VEL
LIN {X 0,Y 156.223,Z 509.865,A -85,B 0,C 180,E1 -23824.554,E2 -23824.554} C_VEL
LIN {X 0,Y 156.406,Z 523.464,A -85,B 0,C 180,E1 -23826.322,E2 -23826.322} C_VEL
LIN {X 0,Y 157.238,Z 535.751,A -85,B 0,C 180,E1 -23828.362,E2 -23828.362} C_VEL
LIN {X 0,Y 158.437,Z 548.231,A -85,B 0,C 180,E1 -23830.905,E2 -23830.905} C_VEL
LIN {X 0,Y 159.472,Z 557.017,A -85,B 0,C 180,E1 -23833.025,E2 -23833.025} C_VEL
LIN {X 0,Y 158.267,Z 568.388,A -85,B 0,C 180,E1 -23836.519,E2 -23836.519} C_VEL
LIN {X 0,Y 157.548,Z 577.942,A -85,B 0,C 180,E1 -23840.15,E2 -23840.15} C_VEL
LIN {X 0,Y 157.293,Z 585.406,A -85,B 0,C 180,E1 -23843.587,E2 -23843.587} C_VEL
LIN {X 0,Y 157.265,Z 592.14,A -85,B 0,C 180,E1 -23847.439,E2 -23847.439} C_VEL
LIN {X 0,Y 157.294,Z 595.831,A -85,B 0,C 180,E1 -23850.001,E2 -23850.001} C_VEL
LIN {X 0,Y 156.99,Z 598.86,A -85,B 0,C 180,E1 -23852.566,E2 -23852.566} C_VEL
LIN {X 0,Y 156.281,Z 603.42,A -85,B 0,C 180,E1 -23857.754,E2 -23857.754} C_VEL
LIN {X 0,Y 156.753,Z 606.626,A -85,B 0,C 180,E1 -23862.955,E2 -23862.955} C_VEL
LIN {X 0,Y 158.636,Z 608.592,A -85,B 0,C 180,E1 -23868.067,E2 -23868.067} C_VEL
LIN {X 0,Y 162.206,Z 609.517,A -85,B 0,C 180,E1 -23872.952,E2 -23872.952} C_VEL
LIN {X 0,Y 167.099,Z 609.365,A -85,B 0,C 180,E1 -23877.559,E2 -23877.559} C_VEL
LIN {X 0,Y 173.314,Z 608.164,A -85,B 0,C 180,E1 -23881.814,E2 -23881.814} C_VEL
LIN {X 0,Y 180.931,Z 605.932,A -85,B 0,C 180,E1 -23885.638,E2 -23885.638} C_VEL
LIN {X 0,Y 189.657,Z 602.627,A -85,B 0,C 180,E1 -23889.048,E2 -23889.048} C_VEL
LIN {X 0,Y 197.763,Z 598.929,A -85,B 0,C 180,E1 -23891.731,E2 -23891.731} C_VEL
LIN {X 0,Y 200.526,Z 597.325,A -85,B 0,C 180,E1 -23893.113,E2 -23893.113} C_VEL
LIN {X 0,Y 202.168,Z 596.296,A -85,B 0,C 180,E1 -23894.106,E2 -23894.106} C_VEL
LIN {X 0,Y 204.33,Z 594.704,A -85,B 0,C 180,E1 -23896.246,E2 -23896.246} C_VEL
LIN {X 0,Y 204.431,Z 594.066,A -85,B 0,C 180,E1 -23899.218,E2 -23899.218} C_VEL
LIN {X 0,Y 204.29,Z 594.118,A -85,B 0,C 180,E1 -23899.288,E2 -23899.288} C_VEL
LIN {X 0,Y 202.242,Z 594.91,A -85,B 0,C 180,E1 -23899.97,E2 -23899.97} C_VEL
LIN {X 0,Y 198.456,Z 596.333,A -85,B 0,C 180,E1 -23900.635,E2 -23900.635} C_VEL
LIN {X 0,Y 189.988,Z 598.982,A -85,B 0,C 180,E1 -23901.713,E2 -23901.713} C_VEL
LIN {X 0,Y 186.845,Z 599.739,A -85,B 0,C 180,E1 -23902.461,E2 -23902.461} C_VEL
LIN {X 0,Y 177.034,Z 601.325,A -85,B 0,C 180,E1 -23906.236,E2 -23906.236} C_VEL
LIN {X 0,Y 169.222,Z 601.554,A -85,B 0,C 180,E1 -23910.108,E2 -23910.108} C_VEL
LIN {X 0,Y 162.576,Z 600.655,A -85,B 0,C 180,E1 -23914.388,E2 -23914.388} C_VEL
LIN {X 0,Y 157.167,Z 598.615,A -85,B 0,C 180,E1 -23919.039,E2 -23919.039} C_VEL
LIN {X 0,Y 153.011,Z 595.413,A -85,B 0,C 180,E1 -23924.004,E2 -23924.004} C_VEL
LIN {X 0,Y 150.31,Z 590.963,A -85,B 0,C 180,E1 -23929.221,E2 -23929.221} C_VEL
LIN {X 0,Y 149.049,Z 585.18,A -85,B 0,C 180,E1 -23934.589,E2 -23934.589} C_VEL
LIN {X 0,Y 148.593,Z 577.648,A -85,B 0,C 180,E1 -23940.001,E2 -23940.001} C_VEL
LIN {X 0,Y 148.718,Z 570.72,A -85,B 0,C 180,E1 -23944.066,E2 -23944.066} C_VEL
LIN {X 0,Y 149.244,Z 562.311,A -85,B 0,C 180,E1 -23948.122,E2 -23948.122} C_VEL
LIN {X 0,Y 150.204,Z 552.103,A -85,B 0,C 180,E1 -23952.156,E2 -23952.156} C_VEL
LIN {X 0,Y 151.449,Z 540.8,A -85,B 0,C 180,E1 -23955.822,E2 -23955.822} C_VEL
LIN {X 0,Y 153.044,Z 528.175,A -85,B 0,C 180,E1 -23959.099,E2 -23959.099} C_VEL
